(* IEC 61131-3 sources: ml2plc/examples/models/structured_text (part 10) *)

    weights_2 : ARRAY[0..587] OF REAL := [0.015340, -0.219861, -0.051065, 0.087872, 0.001123, -0.000694, -0.000503, -0.080889, -0.021135, -0.014471, -0.082583, -0.025172, 0.069586, 0.000587, -0.088471, 0.003759, -0.014212, -0.039110, -0.007912, -0.105317, -0.021763, 0.126463, -0.041350, 0.108134, -0.142301, -0.053275, 0.007500, 0.120579, 0.091133, 0.103068, -0.006133, -0.082495, 0.034790, 0.002800, 0.014254, 0.050135, 0.050392, -0.065882, 0.073643, 0.079869, -0.165370, -0.153988, 0.109092, 0.031460, 0.038941, -0.087463, -0.087233, -0.123573, -0.001647, 0.004770, 0.048463, -0.043877, -0.184602, -0.074370, 0.166586, 0.231821, -0.353194, 0.011201, 0.023368, 0.060943, 0.075272, -0.042498, 0.053250, -0.100004, -0.036177, 0.065228, -0.023655, -0.016418, -0.006418, -0.172362, -0.131650, 0.045625, 0.096511, 0.126555, 0.121202, -0.064907, -0.098812, -0.091086, 0.010892, 0.012223, -0.059166, 0.035979, -0.151760, 0.028790, 0.081683, 0.051266, -0.099853, -0.051092, 0.055367, 0.050935, -0.059011, -0.033349, -0.019745, -0.141106, -0.147728, -0.164434, -0.113353, -0.053255, 0.023697, 0.071369, 0.115603, -0.270532, -0.017005, 0.015443, 0.033358, -0.027488, -0.120684, 0.053873, 0.046257, -0.048391, -0.013597, -0.155116, -0.101134, -0.222254, 0.105084, 0.104957, -0.208010, -0.081657, -0.136778, -0.070762, 0.148919, 0.151061, 0.138501, 0.115350, 0.039400, 0.091898, -0.109483, -0.207599, -0.054447, 0.127668, 0.008047, 0.087241, -0.038910, 0.138434, -0.038079, 0.070282, 0.095658, 0.048807, -0.081151, -0.133361, 0.009412, -0.027122, -0.098228, 0.001431, 0.004148, -0.083694, -0.036905, -0.212899, -0.099266, -0.054151, 0.010881, -0.082305, -0.021167, -0.016677, -0.138309, -0.079492, -0.045268, -0.012169, -0.016324, -0.059901, 0.029291, 0.037319, -0.106169, 0.072890, 0.053698, 0.036590, 0.031903, 0.081211, 0.046060, 0.124919, 0.117014, -0.103158, -0.081969, 0.141857, 0.110490, 0.008438, 0.045665, -0.042151, -0.082792, -0.089687, 0.003011, -0.079598, -0.013750, 0.011140, -0.033389, 0.000607, 0.054720, 0.044793, 0.059433, -0.049758, 0.003480, 0.032585, 0.099914, 0.124206, -0.103656, -0.036959, 0.191891, -0.166580, 0.032615, 0.068289, -0.002894, 0.153752, 0.186112, -0.195345, -0.026172, -0.075779, -0.150166, 0.066905, 0.193295, -0.375487, -0.153804, -0.064015, 0.001013, 0.051095, -0.055609, -0.045019, -0.076890, -0.054708, -0.006689, -0.066367, 0.086120, 0.139797, -0.050011, -0.067812, -0.047263, -0.073355, -0.003271, 0.015706, 0.020044, -0.025812, 0.092713, 0.059356, 0.027340, 0.108126, 0.188838, -0.104976, -0.027165, 0.083738, 0.040041, 0.159310, 0.142973, 0.100962, -0.057635, 0.104709, -0.046478, 0.050873, 0.025351, -0.109376, 0.011739, -0.063282, -0.068576, -0.007735, -0.119382, 0.145221, -0.087949, -0.001548, 0.079334, 0.050926, -0.020037, -0.015313, 0.046571, 0.032091, 0.023714, 0.049098, 0.043621, 0.065767, -0.121593, -0.144732, 0.087293, -0.020124, 0.165755, -0.049488, -0.192976, -0.057565, -0.115345, -0.055495, -0.078657, 0.070386, 0.053267, -0.047640, 0.089666, 0.074974, 0.047833, 0.104152, -0.039127, 0.127704, -0.117635, 0.009256, 0.057764, -0.018319, 0.044890, -0.124445, -0.081869, -0.128226, 0.073160, -0.069937, 0.090754, 0.040999, -0.061193, 0.026409, 0.119392, -0.038913, -0.081897, 0.050141, -0.041159, 0.018876, -0.029160, 0.061441, 0.084635, -0.047072, 0.062523, 0.081736, 0.012864, -0.124673, -0.040521, -0.031922, 0.010283, 0.007151, -0.035083, 0.061101, 0.118654, -0.023953, -0.013829, 0.030714, -0.167063, -0.041738, -0.014768, -0.060637, 0.029150, 0.043681, 0.069267, -0.066030, 0.016060, 0.030191, 0.072170, 0.120849, -0.083327, -0.090694, -0.027987, 0.023541, 0.067148, 0.139641, 0.111992, 0.115982, -0.002341, 0.013067, -0.113392, -0.151181, 0.086295, 0.008997, 0.108310, 0.012295, 0.020733, 0.024920, -0.047194, -0.007393, -0.027599, 0.150969, 0.041255, -0.072869, -0.231603, -0.078684, -0.006606, -0.022358, -0.011507, -0.054861, 0.048565, -0.117770, 0.037562, -0.101887, -0.217231, -0.177524, -0.162331, -0.325387, 0.103984, 0.039200, -0.041771, 0.006172, 0.062825, -0.139174, -0.098610, -0.065995, -0.047678, -0.009318, 0.107075, -0.006649, 0.059119, 0.087902, 0.003926, 0.023742, -0.024262, -0.018050, 0.007341, 0.009480, -0.122970, -0.021484, 0.124687, 0.030027, 0.096136, 0.053442, 0.014279, 0.038727, 0.068228, -0.029878, 0.026607, 0.088246, 0.138748, -0.166321, -0.035119, 0.030434, -0.057495, 0.037143, -0.085420, 0.031156, 0.004837, -0.115455, -0.013989, 0.165773, 0.007360, 0.120774, -0.095685, -0.203753, -0.112300, -0.139024, 0.004306, -0.041803, -0.030506, -0.033363, -0.031449, 0.092906, 0.227986, -0.103965, 0.010845, -0.128290, 0.097496, -0.021628, 0.017594, 0.054620, 0.088933, 0.056891, -0.002936, -0.038590, -0.048186, -0.021997, 0.106340, 0.017138, 0.079845, 0.036567, -0.064192, 0.034146, 0.052743, -0.004024, 0.135401, -0.092349, -0.039482, 0.036607, -0.113198, 0.036544, 0.077170, 0.046460, 0.094072, 0.058304, 0.084231, -0.093658, 0.080444, -0.094438, 0.026712, 0.042926, -0.037896, 0.031974, 0.018030, -0.045118, 0.039413, -0.087483, 0.054411, -0.109296, -0.120550, 0.081438, 0.039630, 0.131441, 0.016337, 0.018872, 0.038904, 0.024723, -0.125727, -0.003417, 0.113643, 0.012522, 0.023285, -0.022591, -0.082088, -0.102981, -0.128956, 0.016828, 0.053169, -0.013050, 0.047433, 0.119200, -0.020646, 0.082886, 0.121989, -0.094658, -0.060755, 0.019658, -0.020039, 0.056247, 0.054539, 0.134044, 0.104659, 0.135269, -0.109605, -0.042843, 0.008803, 0.033988, -0.264132, -0.142610, -0.095774, -0.150958, 0.018190, 0.003449, -0.089845, -0.132400, 0.022324, 0.100510, -0.288181, -0.014459, 0.059133, 0.074987, -0.005254, -0.103758, -0.007229, -0.006405, 0.006130, 0.046741, 0.116869, -0.032138, 0.051615, -0.051291, -0.050372, -0.068670, 0.011227, 0.032439, 0.064744, 0.039815, -0.046261, 0.007456, 0.054653, -0.076340, 0.076204, -0.009191, 0.110411, 0.126815, 0.058138, -0.038349, 0.037423, 0.073164, 0.105311, 0.107432, -0.038734, -0.004818, 0.013107, 0.024137, -0.005680, 0.019150, 0.033298, 0.097045, 0.108157, 0.044789, -0.004634, 0.055465, 0.016219, 0.151309, 0.033116, 0.036895, 0.003101, 0.089325, 0.030543, 0.060574, -0.338772, 0.009696, -0.068708, -0.048821, 0.097889, 0.163710, 0.087727, 0.021977, -0.192762, -0.018846];
    bias_2 : ARRAY[0..2] OF REAL := [-0.598696, 0.937560, -0.406395];

END_VAR

VAR
    (* Buffer allocation variables *)
    buffer_0 : ARRAY[0..195] OF REAL;
    buffer_1 : ARRAY[0..255] OF REAL;

    (* Temporary computation variables *)
    i : DINT;
    j : DINT;
    sum : REAL;
    max_val : REAL;
    exp_sum : REAL;

END_VAR

(* Layer 0: Fused Linear + RELU *)
FOR j := 0 TO 255 DO
    sum := 0.0;
    FOR i := 0 TO 4 DO
        sum := sum + input_data[i] * weights_0[i * 256 + j];
    END_FOR;
    buffer_1[j] := MAX(sum + bias_0[j], 0.0);
END_FOR;

(* Layer 1: Fused Linear + RELU *)
FOR j := 0 TO 195 DO
    sum := 0.0;
    FOR i := 0 TO 255 DO
        sum := sum + buffer_1[i] * weights_1[i * 196 + j];
    END_FOR;
    buffer_0[j] := MAX(sum + bias_1[j], 0.0);
END_FOR;

(* Layer 2: Fused Linear + SOFTMAX *)
FOR j := 0 TO 2 DO
    sum := 0.0;
    FOR i := 0 TO 195 DO
        sum := sum + buffer_0[i] * weights_2[i * 3 + j];
    END_FOR;
    output_data[j] := sum + bias_2[j];
END_FOR;

max_val := output_data[0];
FOR i := 1 TO 2 DO
    IF output_data[i] > max_val THEN
        max_val := output_data[i];
    END_IF;
END_FOR;

exp_sum := 0.0;
FOR i := 0 TO 2 DO
    output_data[i] := EXP(output_data[i] - max_val);
    exp_sum := exp_sum + output_data[i];
END_FOR;

FOR i := 0 TO 2 DO
    output_data[i] := output_data[i] / exp_sum;
END_FOR;

END_FUNCTION_BLOCK

(* ---- test7_6k.st ---- *)
FUNCTION_BLOCK NeuralNetworkFB

VAR_INPUT
    input_data : ARRAY[0..4] OF REAL;
END_VAR

VAR_OUTPUT
    output_data : ARRAY[0..2] OF REAL;
END_VAR

VAR CONSTANT
    weights_0 : ARRAY[0..399] OF REAL := [-0.204252, 0.095494, -0.178736, -0.051593, -0.154857, -0.111379, -0.197264, -0.143097, 0.109827, -0.097160, 0.012020, -0.049268, -0.066065, 0.005468, -0.112784, -0.022716, -0.225224, -0.191850, -0.006850, 0.088268, 0.127013, -0.051319, -0.177738, -0.065624, 0.153682, 0.155821, 0.040109, -0.174692, -0.286252, 0.062215, -0.175209, -0.111276, -0.147501, -0.127080, 0.122492, 0.111213, 0.028250, -0.187593, 0.149308, 0.140091, 0.112817, -0.082366, -0.154004, 0.019695, -0.076321, 0.047790, -0.005837, 0.106352, -0.126226, -0.091414, -0.224965, -0.021193, 0.065960, 0.078478, -0.162489, -0.177320, 0.118103, -0.118781, -0.258763, -0.167764, -0.097012, -0.191475, -0.225075, -0.097829, -0.133086, -0.161308, 0.068450, -0.142950, -0.218535, 0.051961, 0.024169, -0.169507, -0.262286, 0.029901, 0.048540, 0.027806, -0.189779, 0.069045, 0.117139, -0.010558, -0.032235, -0.086801, 0.151290, 0.170069, 0.043408, -0.094498, -0.177663, 0.095259, -0.083921, 0.266576, -0.232399, 0.088012, -0.144461, 0.013028, 0.218332, 0.118870, 0.049978, -0.108692, -0.017786, -0.028464, 0.071001, -0.202678, -0.007252, 0.046975, -0.022387, -0.176915, 0.184037, 0.138823, 0.117583, 0.033052, 0.015849, 0.231544, 0.199028, -0.026578, -0.236188, 0.131210, -0.105877, -0.087975, -0.089525, -0.271682, -0.310378, -0.190208, -0.103984, 0.021078, -0.061623, -0.223657, 0.115391, -0.052116, -0.091774, 0.111931, -0.085383, -0.115295, -0.241702, -0.144102, -0.001192, -0.097169, -0.177709, -0.113947, -0.007674, -0.135584, 0.123896, 0.092379, 0.005358, -0.157152, -0.059988, -0.012534, 0.034736, -0.043048, 0.057696, -0.238518, 0.035371, -0.093588, 0.167829, -0.046709, 0.036370, -0.003444, -0.106658, 0.028076, 0.151991, 0.154167, -0.017135, -0.263429, 0.026569, -0.116189, -0.091898, 0.047045, 0.267170, 0.114090, 0.116855, 0.032118, 0.099443, 0.013459, 0.247495, -0.047596, -0.170523, -0.138334, -0.014806, 0.093128, -0.113583, -0.042853, -0.078199, 0.216203, 0.089752, -0.194084, -0.181997, 0.131227, -0.069781, 0.133463, -0.154973, 0.009000, -0.012056, -0.165474, 0.081740, 0.099855, -0.149436, -0.029881, -0.055397, 0.210030, -0.245871, 0.129955, 0.110984, 0.270213, 0.000066, -0.234064, -0.167355, -0.006196, -0.161614, -0.083333, -0.230470, -0.085398, -0.155489, 0.196806, 0.059367, 0.177773, -0.031812, -0.105303, 0.169684, 0.096922, -0.081472, 0.044204, -0.176394, -0.252753, -0.084089, 0.174208, 0.011128, 0.036618, 0.039985, 0.063442, 0.014899, 0.025740, -0.126109, 0.051767, 0.112909, 0.030818, 0.068933, 0.024684, -0.106318, -0.005054, -0.144284, -0.256852, -0.164291, -0.133206, -0.210012, -0.101632, 0.222082, 0.153257, -0.192512, 0.005971, -0.123604, -0.264094, -0.027056, -0.013892, -0.236922, 0.115783, 0.095674, 0.181820, 0.094948, 0.002586, -0.087751, -0.234015, -0.217941, -0.202149, -0.182678, -0.162661, -0.103708, -0.300429, -0.038539, -0.114616, -0.039287, -0.323055, -0.037187, 0.185280, -0.134350, -0.202214, -0.095785, -0.238161, 0.248820, -0.025541, 0.153553, -0.146549, 0.025226, -0.124733, -0.153933, -0.057788, 0.112253, 0.171774, -0.055901, 0.100347, -0.016596, 0.038081, 0.060529, -0.211000, 0.010525, -0.175179, -0.266535, 0.149374, -0.227717, 0.025317, 0.156851, 0.099082, 0.142311, -0.009360, 0.116468, 0.063573, 0.171788, 0.104363, -0.112531, 0.109297, 0.087755, -0.007313, 0.042170, 0.011677, -0.244264, -0.025654, -0.082018, -0.040680, -0.066031, 0.099246, -0.016522, -0.033168, -0.102887, -0.139828, -0.135602, -0.001694, -0.159093, -0.118193, 0.253445, -0.227600, 0.115132, -0.149348, -0.024129, -0.094190, -0.174122, 0.091905, 0.084444, -0.253624, 0.046840, 0.005839, 0.162217, -0.263061, 0.010626, 0.172488, 0.044317, 0.030137, 0.082965, -0.289103, -0.425034, 0.089364, 0.139634, -0.374789, 0.002438, -0.053035, -0.205200, 0.042774, 0.083738, 0.165071, -0.181691, -0.060783, -0.208866, -0.016353, -0.150721, 0.082961, -0.194339, -0.103480, -0.062981, 0.183148, -0.146493, -0.192516, 0.006207, 0.166178, 0.119890, -0.161796, -0.046662, -0.139639, 0.107740, 0.150401, -0.042296, 0.020544, -0.142547, 0.079611, 0.168141, 0.162479, -0.125809, -0.131995, 0.147326, 0.206230, 0.039064, -0.003743, -0.201281, 0.075811, 0.106736, -0.157088, 0.096469, 0.149164, -0.048443, -0.147991, 0.003754, -0.211540, -0.015394, -0.123360];
    bias_0 : ARRAY[0..79] OF REAL := [0.085009, 0.139520, 0.248067, 1.399861, 0.583598, 0.015434, -0.202390, 0.740568, -0.902567, 0.016522, -0.292847, 1.752811, -0.063338, -0.564435, -1.102493, -0.004024, -0.597225, 0.046091, 0.423281, 0.308277, -0.198749, 0.191307, -0.275388, -0.046908, -0.389957, 0.456703, 0.444849, -0.885773, 0.015246, 0.438173, 0.310576, -1.156887, 0.283457, -0.324643, -0.165189, -0.746600, 0.758963, -0.005614, -0.150126, 0.284105, -0.379746, 0.854058, -0.107690, 0.052858, -0.034767, -0.935268, -0.085336, 1.113907, -0.062266, -0.710800, -0.218181, 0.473975, 0.306379, 0.051084, -0.381713, 0.449957, 0.295188, -0.428395, 0.386686, -0.302978, -0.218029, -0.006667, 0.249048, 0.384831, -1.063448, -0.870574, -0.613569, -0.747093, -0.019498, -0.541172, -1.064162, 0.472992, 0.204574, -0.857920, -0.625336, -0.146532, -0.007889, -0.730171, -0.376830, -0.026634];

    weights_1 : ARRAY[0..4799] OF REAL := [-0.187495, -0.043826, 0.011639, 0.068499, -0.019446, 0.115631, -0.047638, -0.110905, 0.095464, -0.000825, -0.147106, -0.138385, 0.173698, -0.115326, 0.005790, -0.077005, 0.183801, -0.196797, -0.004029, -0.178881, 0.095461, -0.234334, 0.116176, 0.020930, 0.100273, -0.069382, 0.012484, -0.061318, 0.076773, -0.161382, -0.212827, -0.106095, -0.170268, -0.227658, -0.157359, -0.001001, 0.019196, 0.052587, -0.065633, 0.121859, -0.043743, 0.056348, -0.200779, 0.011906, -0.185246, 0.005645, -0.224972, -0.078873, 0.012620, -0.098199, -0.035988, -0.043461, -0.058674, -0.026206, 0.058788, -0.126039, -0.214524, -0.215762, -0.047320, -0.167665, 0.081893, -0.181390, 0.147489, -0.050866, -0.159085, 0.025241, -0.075018, 0.080488, -0.144720, -0.183416, -0.000486, 0.277692, -0.025934, -0.091180, 0.135423, -0.071436, -0.206965, -0.032235, -0.070909, -0.118695, 0.120077, -0.224050, -0.086073, 0.058597, -0.003604, -0.190653, 0.187794, -0.105244, -0.139862, 0.095354, -0.079105, -0.049326, -0.180191, 0.046015, -0.008404, -0.009414, 0.007191, -0.167950, 0.064259, 0.028046, -0.065026, 0.002607, 0.055868, -0.016474, 0.038395, -0.073723, -0.001131, -0.097771, 0.086923, 0.060480, 0.102652, 0.151700, -0.249111, -0.000081, -0.115305, 0.119442, -0.017911, -0.276544, -0.195153, 0.023084, 0.061307, -0.149912, 0.126201, 0.077160, 0.147664, 0.135438, 0.179792, -0.136279, 0.128259, -0.029156, -0.105667, -0.013778, 0.067171, -0.212397, 0.135022, -0.092745, -0.212069, -0.083156, -0.273877, -0.080802, -0.036298, 0.074901, -0.197178, 0.189450, -0.212966, 0.089309, 0.201708, -0.157652, 0.104825, -0.088819, -0.017402, -0.200047, -0.095955, 0.102139, 0.042738, -0.085193, -0.087002, -0.084559, 0.014232, -0.160413, -0.342999, -0.172071, 0.030429, -0.141189, -0.242259, -0.189519, 0.141134, -0.151873, -0.033610, -0.155085, 0.096499, -0.170400, -0.030843, -0.192798, 0.082588, -0.197594, -0.127308, -0.215119, -0.164729, -0.082233, -0.329844, 0.368244, -0.284488, -0.291019, -0.331445, 0.198686, -0.097576, -0.033210, 0.217893, 0.111894, -0.030753, -0.229657, 0.127646, -0.247362, 0.004571, -0.221431, 0.197898, 0.003611, 0.001089, 0.217739, 0.009284, -0.169147, -0.171246, -0.217403, -0.194864, 0.208354, -0.316288, -0.209805, -0.538319, 0.125899, -0.174896, -0.237079, 0.022632, 0.071399, 0.183040, -0.119043, -0.077857, -0.037180, 0.391291, 0.080994, 0.094256, -0.231882, 0.044936, 0.172367, -0.197255, -0.202964, -0.189238, 0.088037, 0.016176, 0.049230, 0.086076, -0.165083, -0.123050, -0.217327, -0.104082, -0.184468, -0.084095, -0.192575, -0.003610, 0.003037, -0.109199, 0.129669, -0.121035, -0.062529, -0.063750, 0.104687, 0.028781, -0.149673, 0.198580, 0.131386, 0.071709, -0.227315, 0.138179, -0.009123, 0.102321, -0.095555, 0.094151, 0.123000, 0.224575, -0.096633, 0.042278, 0.084082, 0.031284, -0.107486, 0.016887, -0.039989, 0.009479, -0.112127, -0.227535, 0.007071, -0.043445, -0.166035, 0.115495, -0.269776, 0.124071, -0.072062, -0.180874, -0.140957, 0.158938, -0.171277, -0.151687, 0.004736, -0.133418, 0.071863, -0.123936, -0.008774, -0.073201, -0.059242, -0.054432, 0.027825, -0.161739, -0.079946, 0.093769, 0.128523, 0.043888, -0.155475, -0.230641, 0.122559, 0.076405, -0.181072, -0.127761, 0.012384, 0.021831, -0.244387, 0.085400, -0.134273, -0.205303, -0.012499, 0.001737, 0.098550, -0.193665, 0.050139, 0.092846, -0.051853, 0.048240, 0.039286, 0.149299, -0.087487, 0.155728, 0.110941, 0.075036, -0.149393, 0.069146, 0.188267, -0.152000, -0.172031, 0.024997, -0.087718, 0.050184, -0.153210, 0.046277, -0.180275, -0.025535, -0.116391, 0.104334, 0.018564, -0.028917, -0.084740, -0.136146, -0.100181, 0.038304, 0.091499, -0.064747, 0.160913, -0.017199, -0.147531, -0.109603, -0.032457, 0.097940, -0.100716, -0.059666, -0.061391, 0.088145, -0.192598, -0.125311, -0.157310, 0.002378, 0.121867, 0.102271, 0.080352, -0.057906, 0.063848, 0.019965, -0.227923, 0.051208, 0.088724, 0.149698, 0.064482, -0.033688, -0.202038, 0.055623, -0.142244, 0.118062, 0.013894, -0.217208, 0.125276, -0.085431, -0.050093, -0.078770, -0.127041, -0.181141, 0.038965, -0.253101, -0.069012, -0.148941, 0.028103, -0.097699, -0.128741, -0.147791, 0.149346, 0.024986, 0.058569, 0.143465, 0.145976, -0.067909, -0.015331, -0.043340, -0.096023, 0.123826, 0.016238, -0.173743, -0.066383, 0.091369, -0.029829, 0.159701, -0.052570, -0.188634, 0.033418, -0.043469, 0.226051, -0.138364, -0.055090, 0.100096, 0.054385, -0.082675, 0.052667, -0.174938, -0.010745, -0.130078, 0.125440, -0.065375, 0.079887, -0.045133, -0.048312, -0.037418, -0.081846, 0.128402, -0.121171, -0.021942, -0.143802, -0.240385, -0.098094, 0.214161, -0.048066, -0.104972, 0.177667, -0.027555, 0.199294, -0.277881, -0.103592, -0.101064, -0.111686, -0.052772, 0.002445, -0.221140, 0.200714, -0.029648, -0.351862, 0.087262, 0.149245, -0.019061, -0.170681, 0.079724, -0.139517, -0.080832, -0.183112, -0.155987, 0.111392, -0.012468, -0.261954, -0.013893, -0.140637, -0.064067, 0.087971, -0.098510, -0.073594, 0.139888, -0.085039, 0.040758, -0.128766, 0.263592, -0.257286, -0.202891, 0.100467, -0.010248, 0.014490, 0.076027, -0.041766, -0.131794, -0.181699, 0.141993, 0.089453, -0.191971, 0.038637, 0.071693, 0.041796, 0.073103, 0.145141, -0.148769, 0.095703, -0.006099, 0.053828, -0.166412, 0.109511, 0.111218, 0.062706, 0.039294, 0.024273, -0.008815, -0.122314, 0.041015, -0.064941, -0.049589, 0.162990, 0.170278, -0.122815, 0.145788, 0.033580, 0.010933, 0.020278, 0.165807, -0.145881, 0.200069, 0.132890, -0.225906, 0.102775, 0.112111, -0.110968, -0.327020, -0.063996, 0.018829, -0.105115, -0.035790, -0.111621, -0.161010, -0.136633, 0.132319, -0.232511, 0.068281, -0.190410, -0.280823, 0.037700, -0.036999, -0.202194, -0.009511, -0.062345, 0.223302, 0.224884, -0.037151, 0.133080, -0.105688, 0.104093, -0.044832, -0.119623, -0.100510, -0.010594, -0.177663, -0.143772, -0.129429, -0.155730, 0.074013, 0.203130, -0.168618, 0.197457, -0.075762, 0.002407, -0.127743, -0.027171, 0.040017, -0.164665, -0.133451, -0.093815, 0.045166, -0.370300, -0.136726, -0.057434, -0.196779, -0.123197, 0.054104, -0.153149, -0.058581, -0.200545, -0.337820, -0.223224, -0.084699, 0.068145, -0.023780, -0.075253, 0.104862, 0.092775, 0.252090, -0.182647, -0.060455, 0.193314, 0.155096, 0.017778, -0.041913, 0.080495, 0.250374, -0.062116, -0.031334, -0.091330, -0.297533, 0.067413, -0.122810, -0.020310, 0.102734, -0.089518, -0.069400, -0.252473, 0.055755, -0.067582, 0.124237, -0.105892, -0.185992, 0.084798, -0.008859, -0.000417, -0.200312, -0.077944, 0.154457, 0.008785, 0.210066, 0.124764, 0.010203, 0.027909, -0.020809, -0.104830, -0.241088, 0.075725, -0.243988, -0.073502, -0.150011, 0.042442, -0.016308, -0.053375, 0.203016, -0.189589, -0.147536, -0.000456, 0.010458, -0.016922, -0.023293, -0.229019, -0.031755, -0.225682, 0.136042, 0.163329, -0.145518, -0.137362, -0.158810, -0.153608, -0.119005, -0.139013, 0.068120, -0.178356, -0.217439, 0.098411, 0.179662, 0.050977, -0.148974, 0.173078, 0.154025, -0.222811, 0.095003, 0.026945, -0.065555, -0.157365, -0.148347, 0.083820, 0.203749, 0.276060, -0.130301, -0.441604, 0.101892, 0.325627, -0.175195, 0.033774, 0.197460, -0.021086, -0.054220, -0.115699, -0.068489, -0.046554, -0.156783, 0.161611, -0.049137, 0.005860, 0.193781, 0.370352, -0.216234, 0.350976, 0.064933, -0.356365, 0.030951, 0.310719, -0.269228, 0.000328, -0.685306, 0.092410, -0.057984, -0.234432, -0.157181, -0.054908, 0.119585, 0.055568, 0.033589, 0.070298, 0.151600, 0.000321, 0.203942, -0.184519, -0.196852, 0.020012, -0.127641, -0.136458, 0.095097, -0.156321, -0.046661, -0.126675, 0.034023, -0.435073, -0.248280, 0.038863, 0.051302, -0.121698, -0.248643, -0.253840, -0.235557, -0.057713, -0.165379, -0.072123, 0.012063, 0.179261, -0.079980, -0.109507, 0.061432, 0.149497, -0.070263, 0.063627, -0.203408, -0.054263, 0.041969, 0.093557, 0.035906, -0.075950, -0.132530, 0.160581, -0.093528, -0.193797, -0.149616, 0.081809, 0.132168, -0.055765, -0.226921, 0.052611, -0.019008, -0.206362, 0.196463, 0.058143, 0.139270, -0.182240, -0.077353, 0.126875, 0.019908, -0.178625, 0.207289, 0.023789, -0.110765, -0.042038, 0.090671, -0.010270, 0.088242, -0.078280, 0.027414, 0.024751, -0.053083, -0.111664, 0.145266, 0.045896, -0.106047, 0.028589, 0.126394, -0.073975, 0.016951, -0.114771, 0.058699, 0.138664, -0.111792, 0.102104, -0.085657, 0.025535, -0.077525, 0.176288, 0.007275, 0.013041, -0.182064, -0.008665, 0.010742, -0.063345, -0.170987, 0.118484, 0.086599, -0.138879, 0.062084, 0.093707, -0.211441, -0.210389, 0.109447, 0.009178, 0.111142, 0.057708, -0.107554, -0.097098, -0.050753, -0.119869, 0.065488, -0.195523, 0.125473, -0.162880, 0.067520, -0.057914, 0.067633, -0.128362, -0.041456, -0.151078, -0.239852, -0.046787, -0.046040, -0.085033, -0.027876, -0.050788, -0.175431, 0.021347, 0.129480, -0.202736, -0.211963, -0.121893, -0.053449, 0.174972, -0.090305, -0.027340, 0.184640, 0.018241, -0.146348, -0.088299, -0.200020, 0.179131, -0.156040, 0.247591, -0.018738, -0.167393, -0.018119, 0.166582, 0.036737, -0.323502, -0.125462, -0.074257, -0.227693, -0.127879, 0.074497, 0.171681, -0.178597, -0.016256, 0.165335, 0.142548, -0.065136, -0.057195, 0.137034, -0.103093, -0.057882, -0.106992, -0.082292, 0.014769, -0.131339, -0.122740, 0.221346, 0.050323, -0.115536, -0.161429, -0.121929, -0.141410, -0.200174, -0.131279, -0.070172, -0.001654, -0.054385, -0.203309, -0.174031, -0.044717, -0.023823, -0.195514, 0.097579, -0.299280, 0.071825, -0.120568, 0.121904, 0.022071, 0.004942, -0.093524, -0.047500, 0.108046, 0.027347, 0.109685, -0.057970, 0.069021, -0.106463, 0.151177, -0.178336, -0.105863, 0.119959, -0.270658, 0.072922, -0.081703, -0.126428, -0.064988, 0.119859, -0.148058, -0.121758, -0.124044, -0.181647, 0.103696, -0.059793, 0.009263, -0.067097, -0.157507, -0.210798, -0.108414, 0.015803, 0.100605, 0.001284, 0.092993, -0.114392, -0.198128, -0.107984, -0.135560, -0.212594, -0.122395, 0.051632, 0.120981, 0.036958, -0.088017, 0.048821, 0.105228, 0.039687, -0.000940, 0.117730, 0.094232, 0.097422, -0.162968, -0.207689, -0.235039, -0.020052, 0.003264, 0.066222, -0.007693, 0.112790, 0.004400, -0.170587, -0.007529, -0.092564, -0.071948, 0.098179, -0.173899, -0.189986, 0.082992, 0.049693, -0.084597, -0.022957, -0.112488, -0.177351, -0.074619, 0.043721, 0.081083, 0.056966, -0.054530, 0.167706, 0.092779, 0.038886, 0.052530, 0.175779, 0.062225, 0.067869, -0.150979, -0.026430, 0.041959, 0.159334, 0.014994, -0.132202, -0.203469, -0.166479, -0.001058, 0.032094, 0.102088, -0.026257, 0.108982, -0.197880, -0.186123, -0.210913, -0.013239, 0.133741, 0.024038, 0.035955, 0.009580, -0.220388, -0.093084, -0.115529, 0.113373, -0.179200, 0.023569, 0.092303, -0.057884, -0.182442, -0.125423, 0.135616, 0.148641, 0.001794, 0.053828, -0.009687, -0.061003, -0.109162, -0.094053, 0.085367, -0.054325, 0.003022, 0.109594, 0.150069, -0.100455, -0.027854, -0.045738, 0.104897, -0.098767, -0.052057, -0.014638, -0.046503, -0.088066, -0.196605, -0.111631, 0.106046, 0.108629, -0.197552, -0.149193, 0.109600, -0.177730, 0.155000, 0.139756, 0.156765, 0.093107, -0.180579, -0.112168, 0.171606, -0.097841, 0.105849, 0.202372, -0.155509, 0.025837, -0.097935, -0.208450, 0.082403, -0.195167, -0.064462, -0.168772, 0.181297, 0.110526, -0.082017, 0.062444, -0.085259, 0.031226, 0.195569, 0.136555, -0.089863, 0.044305, -0.224308, 0.062433, -0.141740, -0.045204, 0.123520, 0.036962, -0.120294, -0.095129, -0.174097, 0.052688, 0.011449, -0.176074, -0.065089, -0.038276, 0.090562, 0.076366, -0.075167, 0.061729, 0.038455, 0.053242, -0.193444, 0.101651, 0.087634, 0.092511, -0.064193, -0.245658, 0.044015, 0.012871, -0.013168, -0.006454, 0.071112, 0.025509, 0.054529, 0.065311, 0.056310, -0.180449, -0.039958, 0.048537, -0.051643, -0.102219, 0.113807, -0.057327, 0.046546, -0.151255, -0.077736, -0.020588, -0.113985, 0.169675, 0.052531, 0.048476, 0.012000, -0.042925, 0.130053, -0.008425, 0.126301, -0.005038, -0.050381, 0.101160, -0.260447, 0.032194, -0.186597, 0.099273, -0.066057, 0.020545, -0.196886, -0.214360, 0.135345, -0.000402, 0.039084, -0.102168, 0.155453, -0.083347, -0.293784, -0.056957, -0.158940, -0.024392, 0.012893, 0.016886, 0.001811, 0.142059, -0.177070, 0.081076, -0.177536, -0.008914, 0.128194, 0.078825, -0.001006, -0.140982, 0.025296, 0.312801, -0.009939, -0.234129, 0.156600, 0.074625, 0.204806, 0.080406, -0.245319, -0.007829, -0.125331, -0.077263, -0.269901, 0.007388, 0.072491, 0.187339, -0.021148, -0.141481, -0.151382, -0.091537, -0.024638, -0.063637, -0.002112, -0.242162, 0.068506, -0.194093, 0.147597, -0.224350, -0.109162, -0.248442, -0.281311, 0.099040, -0.114785, -0.153094, -0.143746, 0.119874, 0.245667, -0.073279, -0.106678, 0.070350, -0.065192, 0.189557, -0.053012, 0.006938, -0.168214, -0.159039, 0.099331, 0.042333, -0.011618, 0.036502, -0.046085, 0.022646, -0.169739, -0.134299, -0.147109, -0.055030, -0.207480, 0.034523, -0.053364, -0.170573, 0.062128, -0.108211, -0.087569, 0.096130, 0.105775, -0.076363, -0.149795, 0.111862, 0.064433, 0.100011, 0.005322, 0.012295, 0.044367, 0.038804, 0.036462, -0.009752, 0.027189, -0.112119, -0.197054, -0.207718, 0.029751, -0.157544, 0.098411, -0.107287, -0.004124, 0.110229, 0.022413, 0.077564, 0.045048, 0.160432, 0.136350, -0.067685, 0.121371, -0.045504, 0.001140, 0.092194, 0.093704, -0.197313, -0.053982, 0.058188, 0.107029, -0.190503, 0.017645, 0.056198, -0.165373, -0.188030, 0.177592, 0.143248, 0.150138, 0.040068, 0.016359, -0.087664, 0.029084, 0.063598, 0.117892, -0.012894, -0.281147, 0.019644, 0.077236, -0.102193, 0.001728, -0.201237, -0.046811, 0.187137, -0.088159, 0.098611, -0.190801, 0.099519, 0.009386, -0.009936, -0.095895, 0.043072, 0.069656, -0.116856, -0.044185, 0.024672, 0.066147, 0.123219, 0.026984, 0.061291, -0.161035, -0.117871, -0.023781, 0.020670, -0.044119, -0.150813, 0.119473, 0.264945, -0.078791, -0.174729, -0.082116, 0.065382, -0.160124, 0.058964, -0.173368, -0.063958, 0.150073, 0.137277, 0.040349, -0.121023, 0.102109, 0.155909, 0.029025, 0.055306, -0.196372, 0.094951, 0.105758, -0.108173, -0.029256, -0.069724, -0.036958, 0.102471, 0.089850, 0.085119, -0.179385, 0.077873, -0.058101, -0.064385, 0.122941, -0.197724, 0.096621, 0.136942, -0.086460, 0.097450, -0.194683, 0.020468, -0.091201, -0.163263, -0.060383, -0.122360, 0.063817, -0.261001, -0.151872, -0.203316, -0.127345, -0.096171, -0.023894, 0.197431, -0.225454, -0.240749, -0.317417, -0.079323, 0.065090, 0.019849, -0.136263, -0.136703, 0.062078, 0.071355, -0.182125, 0.067118, -0.270489, 0.055133, -0.003778, 0.114173, 0.067716, -0.277999, -0.202380, 0.065272, 0.003847, -0.084694, -0.207460, 0.017935, -0.121946, 0.137768, 0.094442, -0.092968, -0.075586, 0.096753, -0.023769, 0.014763, 0.174060, -0.227682, 0.084332, -0.081958, -0.134817, -0.000166, 0.192078, 0.040887, -0.001630, 0.113297, -0.197617, 0.027211, 0.052274, -0.180139, 0.149111, 0.130356, -0.226361, 0.016953, -0.122692, -0.156576, -0.054064, -0.193463, -0.185229, -0.221918, 0.140038, -0.054511, 0.108777, -0.208394, 0.041422, -0.250061, -0.144061, 0.000987, -0.121394, 0.086455, 0.068661, 0.077966, 0.138036, -0.093587, -0.191712, 0.118125, -0.019484, -0.014273, -0.059302, -0.104286, -0.116784, 0.075291, 0.169043, 0.001548, -0.184765, -0.006782, 0.022824, -0.003976, -0.051564, 0.067487, -0.070492, -0.094790, 0.153426, 0.145733, -0.204557, 0.058039, 0.108285, -0.170155, 0.095073, -0.146102, 0.164169, -0.186476, 0.024414, -0.196119, 0.110557, -0.013596, 0.146735, 0.045880, -0.001961, -0.210447, -0.078950, -0.105805, 0.176049, -0.057586, -0.258445, 0.050336, -0.084662, -0.126641, 0.047383, -0.157251, -0.181100, -0.077797, -0.014061, -0.025577, 0.010956, -0.064073, 0.071510, -0.145995, -0.134231, 0.040794, -0.079272, -0.038888, -0.016440, 0.173860, 0.125972, 0.171500, -0.254024, -0.140350, 0.117999, -0.067682, -0.000752, 0.107778, 0.023448, -0.180043, 0.120349, 0.025010, 0.013541, -0.106484, 0.171297, 0.058092, -0.126303, 0.146605, -0.118698, -0.101074, -0.209394, -0.081997, -0.097325, -0.073534, 0.041903, -0.160915, -0.086830, -0.246047, 0.146267, -0.093346, 0.022996, 0.114033, -0.071188, 0.262760, 0.121509, -0.149237, -0.213894, -0.046132, 0.196951, -0.148721, -0.043823, 0.021680, -0.187718, -0.106041, 0.122252, -0.202239, -0.211710, 0.107129, -0.178040, -0.001868, -0.028487, 0.104841, -0.194258, 0.066877, -0.068969, 0.029807, 0.080136, -0.202076, -0.035068, 0.045806, 0.055710, -0.255747, -0.077842, -0.121811, 0.164499, 0.018934, -0.073491, 0.005038, 0.249075, 0.018043, 0.064148, -0.181961, 0.010560, -0.117548, -0.058183, -0.035022, -0.194345, 0.039141, -0.096355, 0.004603, 0.022892, -0.181091, -0.052832, -0.084987, -0.114381, -0.116218, -0.225355, 0.091435, -0.083195, -0.018672, -0.082354, -0.062302, -0.058156, 0.044570, 0.188819, -0.030222, 0.004905, -0.158938, 0.195750, 0.071720, -0.031885, -0.001187, -0.228501, 0.050306, -0.205469, -0.032645, 0.106419, 0.074064, -0.026300, -0.186675, -0.264539, 0.215900, -0.332340, -0.043278, -0.206134, 0.044834, 0.109163, -0.102909, -0.072938, -0.364193, -0.196215, -0.007963, 0.026792, -0.134129, -0.057963, 0.072873, 0.065697, -0.271673, 0.064010, -0.008266, 0.074413, -0.266393, -0.036302, 0.079263, -0.060772, -0.018792, 0.137687, -0.104393, -0.152897, -0.242089, 0.106164, 0.018856, 0.092918, -0.275230, -0.063488, 0.090247, -0.059361, -0.266099, -0.046778, -0.055142, -0.022777, 0.084627, -0.170351, -0.013962, -0.222389, -0.151188, 0.148962, -0.087542, 0.185998, -0.177688, -0.097772, -0.079313, -0.150211, -0.164873, -0.158232, 0.217011, -0.160489, -0.116968, -0.091767, 0.116603, 0.011526, -0.153908, -0.067538, 0.168542, -0.178588, 0.082390, 0.018650, 0.039973, -0.025669, 0.168206, -0.248549, 0.149303, -0.160598, 0.069041, -0.183907, -0.049261, 0.160879, -0.095732, -0.165781, -0.080461, 0.055374, 0.016760, -0.174546, 0.081962, -0.036502, 0.158612, 0.032619, 0.049739, 0.027940, 0.224843, 0.073671, -0.041689, 0.230666, 0.145157, -0.234841, -0.176481, -0.095837, 0.125010, 0.063278, -0.230302, 0.063268, -0.027022, 0.111030, 0.053486, 0.027500, 0.140594, -0.134408, 0.103652, -0.051922, 0.012637, -0.181476, -0.019460, -0.029901, -0.032062, 0.172354, 0.148283, 0.215879, -0.142901, -0.119957, -0.053013, 0.112965, -0.258184, -0.051066, -0.264954, 0.190482, -0.189949, 0.010940, -0.095231, 0.008937, -0.040283, -0.059043, -0.015149, -0.015143, 0.141878, 0.109967, -0.042080, -0.157305, 0.097915, -0.108920, 0.104729, 0.194386, 0.011276, -0.019095, -0.084019, 0.146113, -0.152649, 0.198303, -0.201287, -0.137585, 0.035677, -0.061117, 0.176087, 0.160562, -0.230831, -0.028126, -0.215707, -0.040773, -0.019594, 0.077786, -0.099227, -0.115451, -0.063161, -0.084506, 0.285519, -0.030241, 0.168914, 0.020630, 0.029172, -0.202726, 0.104421, -0.053312, -0.039889, 0.052079, -0.062510, -0.130882, -0.040990, -0.278632, -0.058964, 0.217417, -0.121801, -0.096731, 0.087152, -0.022312, -0.172589, -0.263482, -0.193324, 0.004411, 0.121928, 0.159931, -0.192278, 0.132315, -0.214687, -0.049484, -0.008205, 0.018524, 0.133953, -0.040444, 0.056558, 0.015706, 0.325216, 0.000640, 0.075307, 0.035595, 0.113399, -0.202202, -0.025153, 0.167535, -0.239881, -0.219585, -0.111719, -0.107923, -0.149904, -0.252613, -0.034304, -0.084333, -0.187109, 0.063899, 0.143530, -0.070666, 0.132294, 0.051739, 0.147802, -0.104738, 0.129664, 0.014652, 0.044681, -0.125330, -0.207789, -0.042319, -0.165956, -0.203115, -0.044789, -0.205011, 0.000517, 0.021081, -0.119809, -0.210937, -0.231928, 0.087419, 0.205960, -0.027473, -0.228470, -0.094027, -0.064081, 0.147182, -0.185475, 0.131948, 0.100349, 0.009282, 0.114615, 0.140396, -0.116940, 0.072523, -0.241860, -0.108013, -0.142000, -0.072000, 0.089677, 0.137196, 0.062616, 0.121207, -0.232016, 0.090843, 0.070410, 0.139417, -0.026856, 0.146321, -0.294664, -0.032348, 0.319110, -0.002944, -0.067224, -0.092913, -0.150887, -0.212212, 0.031102, -0.085811, 0.014206, -0.144119, -0.058346, 0.019250, 0.018418, -0.186849, -0.072161, 0.001996, 0.103666, -0.258730, -0.081637, 0.055279, 0.061815, -0.044559, -0.113122, -0.044066, -0.162221, -0.141151, 0.096907, -0.115250, 0.062262, 0.005065, 0.015412, 0.081220, -0.297356, 0.064133, 0.044118, 0.015685, -0.144599, -0.076847, -0.087228, -0.168556, -0.226387, -0.249636, -0.024162, -0.182325, 0.016776, -0.238902, -0.135556, -0.086752, -0.115952, 0.040745, -0.122256, -0.102772, -0.191892, -0.274205, 0.066162, 0.048205, -0.064058, -0.192005, 0.120239, 0.191195, 0.196010, -0.017396, -0.049525, 0.061457, -0.080446, -0.015556, -0.170852, -0.127559, 0.258399, -0.089019, 0.126596, -0.235834, -0.115058, -0.102991, 0.116196, 0.150089, -0.147114, -0.097072, -0.167377, -0.093958, -0.187377, -0.132066, -0.089605, -0.180094, -0.014606, -0.072250, -0.202879, -0.002921, 0.046777, 0.096036, -0.160877, -0.198220, 0.046167, 0.014711, -0.258481, -0.002196, 0.044809, 0.085482, -0.024420, 0.037063, -0.018678, -0.067966, -0.085948, 0.078864, -0.201114, 0.128085, -0.145813, 0.007271, 0.039512, -0.028435, -0.018339, 0.139499, -0.003059, -0.099800, -0.061026, -0.084604, -0.164472, -0.100570, -0.169849, -0.037404, -0.194296, 0.068681, -0.011228, 0.059797, 0.134118, -0.200450, 0.131266, 0.008578, -0.032415, 0.125618, -0.183185, -0.186559, -0.059436, 0.039473, -0.133920, -0.179227, 0.156785, -0.167550, -0.090492, 0.055735, 0.129721, -0.109047, 0.164852, 0.055422, 0.065316, -0.189822, 0.012060, -0.117954, 0.014381, 0.158313, -0.189159, 0.142768, -0.144892, -0.116591, -0.005984, 0.124853, -0.026583, -0.166240, -0.083795, -0.123045, 0.122757, -0.037477, 0.092098, -0.148620, 0.038476, 0.152449, -0.098045, -0.094949, -0.145768, 0.081120, 0.032547, 0.132474, 0.135196, -0.257294, -0.163471, -0.075842, 0.216315, 0.079247, 0.066841, -0.054610, 0.080234, 0.023575, -0.091794, -0.154834, -0.053194, -0.028051, -0.130317, -0.114688, -0.102097, -0.054053, 0.071980, -0.149434, -0.025769, -0.159231, 0.136723, 0.069798, -0.142915, -0.204482, 0.013283, 0.165752, 0.048956, -0.071522, 0.014189, -0.034166, 0.140926, -0.063779, -0.189843, -0.093377, 0.089115, -0.053616, -0.139420, -0.037278, 0.143302, -0.117698, -0.054848, 0.127853, 0.055342, 0.152365, -0.160254, -0.059313, 0.100204, -0.156020, -0.004533, -0.169456, 0.076558, 0.115337, 0.033748, -0.130311, 0.001136, -0.053222, -0.189011, -0.052963, -0.170158, -0.044768, -0.229454, -0.088228, 0.161163, -0.254016, -0.079255, 0.109965, -0.044888, 0.111780, -0.214687, 0.055047, -0.118845, -0.152920, 0.182037, -0.064142, -0.169884, -0.003040, -0.184904, -0.064518, 0.088405, -0.147685, 0.088867, -0.048795, -0.109284, -0.187385, 0.202099, -0.078681, -0.135884, 0.066514, -0.027167, -0.049248, 0.013263, 0.001392, 0.114698, 0.153221, -0.056513, 0.110682, -0.002497, 0.033449, 0.093565, -0.013117, 0.192191, 0.155546, 0.047371, -0.140575, -0.127799, -0.017932, 0.113502, -0.065293, -0.165022, -0.168184, -0.210941, 0.011351, -0.077979, -0.032503, -0.211552, 0.114545, -0.002053, 0.099328, -0.012842, -0.041377, 0.011279, -0.033605, 0.080875, 0.134533, 0.134824, -0.148507, -0.144622, -0.128805, -0.022675, 0.114730, 0.066712, -0.066104, 0.027683, -0.008968, 0.165856, -0.105824, 0.166434, 0.188111, -0.110221, -0.230624, -0.142589, -0.026202, -0.129956, 0.042155, 0.077495, 0.151450, -0.172573, -0.138375, 0.058228, 0.143052, -0.003161, -0.229277, -0.063510, -0.143647, 0.146517, -0.045903, -0.177465, -0.110375, -0.034529, 0.170249, -0.050045, -0.115385, 0.174185, -0.046401, 0.002193, 0.028995, -0.271681, 0.218660, 0.126515, -0.230110, 0.000361, -0.160436, 0.005971, -0.344556, 0.131244, -0.051877, -0.006286, 0.057548, -0.068816, 0.211492, -0.095057, -0.199010, 0.054005, -0.149013, -0.353793, -0.120430, -0.039355, -0.024089, -0.194303, -0.085727, 0.117557, 0.040830, -0.063834, 0.093352, 0.110169, -0.024051, 0.009023, -0.119322, -0.203330, -0.208702, -0.160522, -0.129267, -0.150143, 0.045876, -0.129271, 0.162690, 0.006713, -0.162987, -0.220998, 0.083108, 0.026168, -0.251240, 0.018553, -0.104916, -0.188408, -0.007697, -0.057978, -0.160972, -0.160025, -0.067211, -0.145218, -0.190131, 0.092764, 0.025449, -0.167894, -0.229953, 0.064689, 0.075397, -0.209588, 0.107188, 0.089073, -0.080405, 0.031624, 0.131544, -0.102374, 0.039610, 0.105508, -0.203861, 0.120127, 0.092031, 0.120020, 0.008069, -0.269261, 0.129556, -0.175342, 0.179533, 0.181329, -0.048755, -0.094702, -0.099701, -0.032849, -0.168873, 0.007508, -0.204996, -0.098034, 0.123244, -0.072101, -0.006969, -0.012494, 0.101649, -0.094537, 0.168231, -0.089403, -0.032065, 0.038520, -0.102243, 0.078368, -0.003533, 0.201117, 0.147341, 0.000962, 0.137667, -0.099660, 0.112765, 0.165554, -0.003054, -0.046399, 0.037375, -0.082632, -0.053002, 0.006530, -0.115165, -0.218031, 0.146812, -0.045703, -0.047095, -0.187636, -0.248226, 0.008975, -0.035089, -0.247149, 0.010909, -0.141086, 0.033582, 0.046870, 0.026986, -0.162250, 0.181453, -0.079880, -0.125142, 0.035112, -0.221431, -0.031269, -0.033955, -0.182166, -0.073946, 0.029919, -0.017677, 0.102744, 0.050007, 0.203223, -0.050583, -0.154773, 0.094398, 0.172041, -0.025008, -0.071187, -0.051416, -0.132822, -0.214228, -0.123545, 0.020750, 0.118510, -0.267256, -0.151250, -0.064021, 0.136177, 0.075619, -0.052630, -0.220219, 0.104414, -0.104515, 0.100698, 0.024376, 0.031545, -0.019857, 0.184470, -0.023951, 0.201691, -0.048933, -0.050628, -0.106438, -0.144221, 0.085044, -0.061666, -0.003440, 0.114548, -0.113571, -0.063113, -0.149883, -0.231086, 0.168807, 0.189000, -0.100231, -0.212070, 0.023967, -0.116457, -0.106547, 0.092277, -0.046945, 0.079230, -0.178069, -0.154461, -0.228762, -0.182785, -0.139319, 0.075915, 0.139459, -0.015411, -0.203283, 0.015147, 0.066272, -0.099117, -0.096452, 0.086900, -0.136055, 0.142824, -0.116338, 0.025016, -0.158700, 0.022083, 0.143109, -0.158336, 0.067653, 0.020425, 0.115204, 0.148361, -0.093780, 0.024555, 0.084137, -0.177413, 0.008700, 0.072282, -0.050387, 0.181537, 0.064798, 0.020360, -0.025410, -0.129684, 0.172169, 0.133576, -0.038328, -0.039753, -0.100537, -0.188232, -0.104797, 0.009509, -0.160821, -0.136193, 0.187715, 0.080495, 0.142507, -0.112630, 0.018149, -0.043601, -0.005145, 0.101457, 0.023155, -0.144749, -0.199948, -0.211947, -0.062993, -0.078606, 0.110997, -0.143283, 0.039227, 0.089242, -0.215382, 0.089589, 0.220947, 0.069715, -0.241524, -0.186060, 0.016640, -0.106317, -0.014027, -0.079524, 0.109182, 0.076188, -0.198620, -0.168251, -0.162477, 0.043841, -0.052630, -0.076567, -0.092701, 0.078072, 0.021543, 0.172751, 0.135313, 0.147821, 0.132467, -0.167929, -0.088592, 0.162098, -0.148587, 0.048029, -0.249911, 0.016675, 0.233101, -0.081811, 0.238881, 0.106396, 0.091837, -0.200439, -0.104207, -0.054120, 0.148718, -0.062928, -0.263816, -0.137687, 0.106893, 0.046282, 0.116825, 0.060096, -0.199340, -0.001481, -0.032136, 0.182016, -0.020477, 0.068802, 0.093807, -0.007107, 0.016390, -0.038848, -0.003995, -0.017074, 0.141418, 0.103226, -0.058193, -0.037460, -0.103801, -0.191240, 0.158296, -0.209071, 0.000973, 0.142015, -0.257622, -0.168149, -0.198492, 0.049495, 0.168498, -0.278393, 0.060121, -0.050809, 0.046848, 0.039852, 0.077347, 0.122856, -0.180872, 0.131647, -0.028642, 0.080471, 0.119349, 0.107144, 0.239806, -0.157665, -0.115875, -0.056992, 0.127495, 0.081902, -0.213950, 0.103815, -0.242172, -0.144274, 0.204785, 0.128645, -0.114874, 0.038003, 0.089306, 0.066272, -0.054892, -0.101228, 0.088170, 0.085930, -0.037906, 0.066707, -0.031384, -0.148178, -0.204148, -0.030258, -0.044266, 0.092554, -0.128923, 0.128254, -0.207565, -0.121365, 0.161021, 0.055441, 0.132810, -0.078076, -0.122189, 0.075973, 0.083530, 0.084315, -0.045538, 0.094101, -0.150394, 0.120926, 0.023058, 0.024018, 0.048490, -0.127737, -0.190660, 0.113682, 0.027284, -0.174501, 0.031990, 0.081054, -0.079009, -0.018344, -0.105399, 0.074602, -0.161182, 0.090526, 0.145769, -0.263158, 0.051536, -0.074488, -0.212269, -0.145064, 0.146161, -0.129024, -0.046608, -0.190778, -0.030772, -0.162515, 0.077865, -0.198759, -0.182206, 0.085732, -0.283933, -0.093270, 0.085093, 0.064581, 0.178087, 0.062132, -0.104943, -0.265024, 0.112701, 0.086531, -0.123810, -0.249047, -0.256520, 0.028357, -0.152399, -0.022150, -0.076901, -0.018218, -0.046563, -0.061145, -0.142526, -0.105981, -0.162923, -0.035189, -0.063013, 0.064950, 0.162953, -0.191534, -0.149038, 0.032344, -0.063380, -0.117506, -0.245808, 0.091629, -0.017261, -0.073465, -0.045410, 0.007090, 0.034745, 0.008076, -0.132518, -0.156898, -0.077817, 0.203200, 0.033604, -0.031922, 0.105459, -0.097677, 0.159753, -0.130119, -0.004635, 0.053019, -0.111458, -0.045096, 0.090431, -0.238046, -0.019331, -0.198789, -0.099207, -0.081391, -0.030734, -0.183423, 0.090616, 0.041235, 0.010797, -0.086633, -0.075456, -0.250842, -0.198288, 0.069771, -0.028523, -0.095769, -0.110560, 0.000893, 0.000040, -0.051924, -0.048272, -0.229717, 0.161767, -0.055050, -0.092417, 0.124414, 0.032945, -0.071673, -0.067353, -0.099497, -0.057776, -0.124306, 0.037371, 0.000361, -0.258351, -0.176557, 0.065653, 0.146299, -0.139200, -0.158257, 0.030842, -0.003725, -0.202649, 0.008102, -0.057356, 0.073134, 0.008535, -0.129729, -0.051063, -0.038931, -0.027468, -0.106782, -0.001024, -0.116288, -0.180409, -0.034534, -0.073670, 0.005906, 0.058219, 0.166522, -0.102660, -0.098151, -0.127832, -0.028517, -0.060918, -0.113861, -0.046391, 0.024097, -0.000475, -0.161964, -0.109885, -0.129191, 0.021787, 0.225193, 0.007721, 0.061646, -0.035113, -0.134712, 0.052947, -0.080252, -0.218266, 0.138702, -0.150738, 0.059385, 0.138550, 0.064942, -0.007138, -0.112035, 0.204377, -0.129377, -0.021014, 0.149506, -0.001235, -0.077465, -0.160133, -0.117720, 0.092737, -0.029005, 0.174047, -0.274779, -0.250030, 0.078172, -0.090331, 0.042961, -0.205316, 0.046367, -0.056894, -0.173929, 0.076132, -0.147334, -0.039802, -0.266360, -0.284472, -0.015277, -0.217796, 0.034299, 0.030395, 0.000070, -0.014245, -0.205233, 0.016903, -0.048655, -0.151058, 0.114937, 0.057784, 0.038171, -0.219878, 0.079477, 0.097282, -0.021168, -0.081827, 0.088759, -0.058871, 0.070619, -0.205786, -0.067125, 0.106157, -0.062420, -0.136652, -0.180082, -0.065296, -0.286946, -0.321869, 0.017554, 0.089872, -0.105208, 0.044293, 0.248013, -0.173252, -0.109481, 0.202816, -0.014991, 0.124017, -0.067284, -0.023998, 0.088478, 0.101868, 0.081817, 0.209412, -0.018781, -0.172477, -0.164562, 0.200007, 0.056884, 0.106272, -0.182880, -0.123781, 0.063267, -0.230638, -0.019055, -0.205419, 0.197541, -0.198720, -0.182181, 0.110510, -0.084713, 0.065407, -0.049739, 0.156435, -0.224698, 0.094290, 0.014365, -0.190435, 0.126705, -0.059463, 0.057626, 0.069520, -0.047589, -0.157757, 0.138826, 0.176764, -0.288364, -0.024494, -0.205077, 0.019677, -0.138235, 0.125638, 0.014956, -0.232807, -0.061307, 0.082854, -0.175044, 0.031433, -0.183093, 0.093276, 0.027900, -0.209902, 0.159516, 0.129424, 0.132976, 0.040934, 0.128310, -0.115805, 0.160791, 0.200437, 0.120027, -0.169269, 0.001254, -0.122004, -0.111766, -0.116197, 0.107472, 0.124729, -0.004954, -0.095255, 0.073652, 0.004850, -0.178254, 0.195797, -0.031146, -0.259319, -0.115599, -0.063144, -0.061969, 0.149608, -0.014443, -0.213948, 0.008068, 0.144077, -0.143199, -0.070661, -0.090459, 0.122777, -0.055731, 0.107613, -0.023732, 0.020959, 0.093576, -0.187325, 0.074573, 0.007694, 0.117199, 0.041512, -0.216200, -0.130893, -0.149750, 0.028815, -0.030344, -0.116414, -0.317162, -0.040079, 0.242659, -0.023888, -0.066037, 0.052766, -0.005770, 0.050451, -0.208458, 0.191133, -0.078927, -0.090132, -0.181439, 0.017455, -0.037453, -0.011490, -0.059334, -0.032730, -0.006085, -0.063982, -0.026299, 0.109608, -0.084109, -0.012514, -0.013087, -0.065923, 0.004334, 0.010522, -0.033329, -0.109663, 0.254545, 0.172810, -0.163591, 0.120675, -0.145430, 0.151358, -0.078560, -0.037670, -0.154208, 0.069605, -0.067404, -0.119043, 0.032602, 0.079160, 0.016203, -0.089354, -0.060417, -0.162385, -0.212389, -0.221961, 0.068451, -0.107366, -0.121543, -0.101876, 0.016305, 0.125544, -0.033034, -0.040435, -0.076167, 0.195144, 0.068947, -0.065570, -0.105697, -0.124721, -0.109227, -0.083588, 0.099832, 0.003592, -0.160067, 0.003259, 0.041199, -0.083822, -0.132558, -0.256203, -0.182740, 0.001317, -0.137657, -0.082421, 0.046106, 0.120890, 0.025548, -0.126929, 0.107434, 0.019413, 0.090971, -0.067734, 0.123079, 0.127130, -0.161999, -0.005005, 0.048149, -0.023897, -0.270545, -0.111089, 0.004118, 0.033362, -0.027953, 0.054008, 0.152816, -0.201762, 0.021524, -0.123197, -0.073559, 0.000524, -0.091507, -0.106242, 0.050329, -0.108801, -0.101153, -0.064999, -0.002875, 0.039322, -0.107689, -0.154053, -0.202276, -0.040283, 0.089812, 0.114359, -0.107079, -0.124529, -0.001914, -0.104789, -0.121565, -0.198390, -0.099632, -0.006911, -0.045216, -0.029867, 0.030992, -0.083115, -0.039788, 0.017990, 0.004738, -0.146365, 0.212923, 0.018532, -0.198817, -0.014912, -0.021895, 0.056025, 0.134704, 0.052262, 0.077839, -0.074575, -0.030728, 0.051926, -0.134101, -0.065329, 0.095441, 0.005362, -0.320066, -0.031660, 0.185336, -0.185066, -0.244708, -0.041238, -0.240934, 0.289305, 0.085717, 0.070756, -0.281231, -0.121665, 0.017694, 0.043168, 0.018245, 0.117926, -0.134891, 0.173788, -0.016483, 0.074033, 0.297291, -0.077766, -0.096016, -0.143047, 0.054483, -0.159745, -0.015035, -0.079806, -0.192738, -0.229282, -0.033435, -0.210121, -0.120133, 0.081383, 0.028186, -0.233440, -0.005699, -0.141221, 0.161547, 0.060737, -0.041088, -0.145830, 0.006742, -0.148999, 0.135203, 0.102135, -0.238380, 0.122228, 0.041691, -0.162923, -0.041621, 0.034483, -0.072151, -0.106803, -0.070408, -0.161970, 0.014867, 0.027113, -0.124863, -0.136033, -0.094630, -0.129611, 0.053116, 0.009706, -0.195417, -0.151510, -0.067206, 0.139619, 0.139601, 0.034085, 0.056369, 0.079887, -0.058680, 0.139363, -0.165965, -0.116522, -0.065965, 0.161519, -0.058847, 0.010203, -0.180771, -0.010577, -0.093030, 0.129600, 0.164807, -0.038184, -0.152913, -0.150552, -0.034221, -0.080638, -0.145570, -0.164487, -0.153948, -0.123227, -0.136960, -0.182059, -0.143404, -0.190808, -0.041683, -0.101558, -0.205040, 0.106900, -0.119287, 0.062814, -0.006110, -0.051024, -0.154184, -0.103544, -0.112718, -0.038922, 0.215685, -0.091556, 0.110361, -0.118157, -0.128787, 0.085860, -0.296992, 0.088935, -0.117518, 0.076616, -0.241626, -0.151477, 0.257687, -0.197329, -0.074681, -0.111951, 0.084828, -0.143288, 0.031309, -0.118217, -0.294245, -0.193350, -0.042170, -0.051293, -0.056437, -0.097944, -0.068279, -0.082731, -0.115753, 0.102119, 0.128756, -0.128144, 0.023206, 0.053891, -0.317280, -0.090716, -0.048617, -0.201192, 0.030243, 0.006836, 0.008797, 0.170371, -0.113556, -0.150117, -0.184408, -0.039981, 0.085722, -0.163927, -0.088385, -0.135078, 0.120191, -0.026627, -0.042047, 0.050042, 0.131262, 0.035964, 0.166282, -0.128620, -0.198723, -0.217690, -0.040826, 0.102168, -0.020908, -0.013998, -0.224456, -0.218090, -0.147928, 0.118010, 0.106042, -0.028700, 0.235288, -0.180627, -0.198808, -0.249863, -0.064488, 0.017811, 0.166005, -0.213845, 0.138073, -0.153009, 0.141843, -0.051419, -0.075694, -0.226131, -0.041074, -0.207081, 0.040820, -0.064222, -0.028781, 0.168728, 0.101631, -0.161025, 0.093556, -0.202608, 0.108386, -0.153070, 0.192274, -0.145241, -0.000211, 0.236275, -0.087635, -0.151944, -0.028237, 0.198736, -0.024313, -0.087090, -0.097063, -0.121538, -0.099224, 0.134001, -0.174923, 0.151579, -0.053231, -0.247944, -0.088981, -0.211388, -0.063122, -0.018182, 0.168559, -0.169690, -0.055651, 0.025104, 0.185304, -0.144953, -0.049440, 0.119042, -0.046729, -0.055920, 0.180785, -0.090310, 0.157958, -0.117315, 0.043618, -0.134080, 0.056683, -0.077463, -0.241500, 0.129426, -0.142416, 0.023727, 0.108929, -0.008048, 0.172686, -0.132356, -0.196406, -0.184002, 0.210628, -0.238060, -0.089066, 0.114596, 0.153111, 0.194562, 0.161066, -0.035873, 0.036367, -0.155359, 0.100467, -0.026104, 0.356755, -0.082889, 0.026330, -0.048655, -0.118040, 0.029410, -0.169095, 0.000227, 0.103414, 0.181038, -0.095122, -0.093822, 0.081849, -0.091800, 0.081307, 0.068839, -0.082793, -0.111909, 0.114605, 0.013529, 0.014640, -0.110074, 0.100217, -0.050205, 0.122569, -0.025452, -0.140571, -0.102917, -0.259463, -0.041072, 0.286599, -0.108083, 0.061381, 0.046828, -0.140044, 0.062607, 0.055307, -0.086436, -0.228696, 0.050932, 0.117816, 0.102888, -0.166034, 0.226874, 0.022948, -0.109273, -0.160216, 0.047745, 0.172978, 0.058415, -0.126457, -0.043911, 0.017664, 0.007508, 0.072441, 0.103484, 0.085472, 0.019245, -0.137672, 0.061656, 0.124268, -0.181649, -0.003858, 0.013738, 0.008420, 0.043954, 0.048462, -0.140401, -0.031369, 0.051175, -0.147290, -0.226342, -0.100782, -0.147707, 0.129768, 0.119781, -0.055445, -0.100545, -0.073053, 0.085573, -0.074556, -0.105671, -0.036404, -0.072882, 0.075968, 0.063639, -0.194386, -0.122092, -0.002620, -0.022566, -0.133343, 0.162517, 0.050876, -0.199029, 0.188501, 0.167689, -0.071162, 0.118603, 0.109654, -0.110553, 0.138290, 0.142590, -0.102962, 0.045384, 0.012512, -0.102174, -0.140773, -0.094162, 0.010323, 0.155468, -0.142019, -0.097794, -0.137002, -0.212146, 0.207217, -0.017213, 0.002942, 0.034605, 0.107504, 0.150266, -0.129505, 0.192782, -0.028705, -0.202198, -0.147815, -0.153301, 0.174837, 0.060969, 0.128735, 0.105888, 0.073072, 0.088999, -0.002995, -0.193849, -0.173289, 0.083937, -0.146552, 0.142054, -0.139680, -0.000768, -0.076366, -0.059695, 0.032080, -0.010387, 0.051921, -0.102333, -0.071009, 0.175738, -0.134685, -0.134976, -0.095431, 0.205827, -0.073887, 0.094985, -0.191911, 0.164504, -0.086110, -0.108445, 0.061845, 0.162021, 0.028200, 0.119438, -0.245631, 0.091793, 0.114317, -0.021548, 0.107032, 0.038590, 0.093562, -0.205856, 0.118910, -0.084905, 0.021004, -0.198377, -0.234301, -0.211129, 0.070893, 0.022674, -0.051338, 0.153045, -0.149085, -0.122123, 0.079959, -0.204106, -0.200147, 0.090186, 0.084070, 0.131274, -0.088271, 0.169127, -0.101847, 0.176898, 0.156308, 0.027733, 0.075918, -0.044774, -0.035376, 0.027992, 0.050958, -0.174579, 0.092923, -0.093785, -0.139114, -0.086600, -0.116225, 0.079024, -0.074963, -0.027205, 0.063837, -0.077457, 0.097615, -0.170624, -0.204657, -0.174123, 0.252476, -0.037762, -0.003866, -0.066153, 0.032779, -0.063880, 0.102435, -0.165147, 0.003097, -0.019100, 0.193608, 0.024472, 0.017538, 0.040808, -0.101324, -0.124583, -0.220176, -0.176091, -0.236821, 0.080546, -0.147749, -0.021607, -0.064803, -0.108025, 0.158381, 0.062731, -0.012334, -0.053412, -0.167796, -0.192720, -0.003843, 0.094745, -0.155300, 0.099702, -0.084310, -0.010902, 0.030403, -0.033079, 0.012516, -0.123602, -0.057762, 0.091336, -0.052454, 0.047064, 0.102744, 0.021584, -0.068199, -0.177980, -0.174477, 0.108816, 0.072409, -0.097811, 0.006908, 0.109265, 0.069252, 0.082388, -0.013773, 0.083408, -0.123182, 0.143093, -0.027379, 0.216197, 0.204592, -0.202415, -0.173952, -0.049781, -0.209224, 0.207557, -0.108861, 0.012178, -0.180074, -0.204747, 0.012663, -0.117213, -0.078747, -0.232379, -0.082473, 0.222548, -0.076128, 0.017688, 0.185962, 0.059833, 0.070901, 0.145850, 0.166014, -0.001596, 0.174953, 0.097180, -0.047201, 0.140861, -0.002166, -0.015422, 0.082614, 0.018298, -0.158532, -0.081273, 0.026782, 0.010039, 0.014152, -0.113708, 0.021807, -0.006415, 0.134055, -0.024455, 0.166605, 0.119609, -0.240276, 0.011147, -0.070938, -0.001916, -0.190984, -0.020498, 0.049692, 0.119988, 0.012101, -0.079877, 0.104347, 0.115889, -0.000701, -0.000200, -0.116832, -0.053406, 0.127320, 0.123170, -0.223954, 0.077958, 0.000277, 0.190590, 0.119747, 0.106785, 0.065563, 0.016657, -0.069956, -0.145500, -0.127351, -0.048157, -0.251979, 0.125064, -0.110993, 0.078520, -0.005572, -0.201606, 0.109670, -0.176686, 0.156523, 0.133993, -0.091991, 0.168931, -0.148177, -0.050699, -0.120765, -0.139533, 0.058259, 0.140237, 0.092177, -0.165459, -0.171207, 0.156731, 0.010243, -0.049143, -0.198165, 0.058386, -0.002632, -0.010948, -0.065568, -0.082094, 0.111951, -0.213757, -0.177344, 0.045442, 0.009229, -0.081340, -0.063801, 0.186457, 0.136439, -0.109015, 0.086114, 0.111018, -0.081917, -0.077104, -0.197834, -0.215515, 0.045228, -0.149443, -0.175919, 0.159206, -0.214795, 0.049048, -0.150895, 0.177309, -0.133976, -0.049341, -0.101059, -0.035851, -0.128504, 0.057545, 0.148281, -0.165562, 0.097207, 0.138636, -0.172084, -0.049035, -0.149735, 0.085481, -0.005862, 0.022614, -0.301166, 0.073367, 0.035003, -0.048621, 0.069253, 0.041897, -0.004374, 0.075960, -0.060290, 0.138160, 0.120225, 0.085650, -0.208537, 0.096014, 0.044026, 0.042850, 0.103294, 0.101432, 0.030810, -0.296734, -0.137424, 0.143252, 0.145805, -0.086185, 0.120815, -0.035621, 0.022993, 0.133212, -0.172715, 0.113733, -0.170444, -0.036648, 0.122507, -0.022651, 0.110245, 0.164986, -0.102638, -0.163859, -0.129321, 0.024643, -0.008650, 0.003262, 0.188762, -0.044951, -0.100630, 0.129388, 0.057905, 0.111092, 0.097379, 0.180758, -0.122092, -0.061474, 0.097122, -0.016703, -0.092755, -0.217754, -0.209254, 0.169666, -0.168835, 0.120574, -0.075259, -0.146628, 0.023180, -0.181881, -0.070199, 0.201167, -0.086352, -0.033172, 0.029317, -0.147238, -0.169502, 0.026048, -0.126043, -0.150882, -0.246272, -0.086376, 0.114050, -0.037291, -0.077498, 0.131446, 0.134411, -0.065761, 0.052115, -0.103191, 0.036951, -0.105550, -0.174234, -0.113685, 0.169620, -0.111003, -0.190180, -0.070703, -0.011564, 0.170409, -0.213383, -0.093098, -0.001624, 0.128783, 0.108914, -0.304261, -0.043003, 0.030753, 0.004043, -0.094789, 0.165093, 0.031420, 0.103349, 0.053297, -0.224531, -0.036606, 0.016023, -0.229925, 0.018866, -0.094369, -0.004789, -0.117526, -0.017096, 0.166951, 0.041755, -0.016534, 0.032813, -0.079353, -0.091808, -0.141489, 0.000641, 0.014971, -0.044141, -0.172049, -0.077523, 0.106444, -0.053978, -0.140208, -0.167674, -0.057589, 0.031635, 0.051585, 0.228365, -0.278278, 0.005538, -0.040600, -0.008821, -0.229175, -0.150135, -0.048334, -0.063206, -0.176003, 0.017721, 0.280622, 0.036771, 0.028169, 0.035114, 0.173123, 0.015005, 0.026818, 0.013097, 0.174614, -0.055922, 0.049859, -0.079898, -0.094391, -0.148679, 0.104692, 0.092321, -0.096423, 0.169699, 0.076722, -0.191469, -0.095258, -0.112098, -0.109355, -0.155259, 0.060463, 0.039525, -0.048619, -0.098098, -0.039907, -0.006702, -0.148284, -0.126526, 0.021500, -0.052005, -0.143786, 0.104853, -0.211339, 0.014862, -0.028785, -0.077053, -0.218324, 0.112712, -0.070995, -0.094271, -0.060391, -0.202425, 0.002345, -0.030716, -0.146052, 0.001556, -0.164822, 0.037714, -0.072036, -0.161283, -0.130253, 0.057649, -0.001839, 0.047250, -0.058188, 0.014529, -0.228346, 0.225228, -0.023914, 0.133087, 0.086785, -0.038637, 0.056942, -0.125695, 0.081435, -0.067135, 0.205670, 0.027072, -0.091504, -0.204132, 0.043087, 0.082807, -0.095363, 0.184644, -0.216296, 0.080196, -0.061449, 0.048607, -0.191740, -0.084450, -0.225042, -0.136752, -0.167331, -0.001254, -0.101233, -0.008365, 0.126993, -0.073219, -0.113536, 0.073879, -0.098733, 0.172418, -0.198177, 0.192814, -0.122041, -0.060191, -0.014931, 0.163615, 0.067764, -0.245190, 0.178596, -0.136161, -0.044688, -0.142136, 0.182072, 0.069366, 0.028530, -0.070855, -0.174058, -0.020019, 0.118313, 0.147296, 0.010455, -0.009949, -0.016825, -0.202637, -0.092267, 0.178319, 0.056175, -0.129320, 0.100304, -0.182421, -0.058295, 0.101226, -0.040390, -0.163760, 0.140207, -0.183046, -0.084880, 0.045066, -0.133398, -0.018702, -0.007750, 0.182355, 0.032732, 0.052878, -0.055891, -0.242827, -0.185519, -0.177503, -0.027939, 0.044171, 0.150245, -0.014234, 0.112920, -0.138517, 0.026886, 0.002449, -0.065427, 0.118718, -0.156467, 0.016188, 0.045635, -0.073365, -0.104475, -0.000712, 0.089148, 0.064683, -0.087668, 0.072877, -0.062352, 0.164486, -0.179810, 0.150326, 0.034267, 0.083289, -0.135315, -0.078507, 0.114422, -0.139795, 0.072093, 0.045491, 0.071670, -0.095322, -0.025386, 0.045614, -0.045319, 0.027453, -0.017968, 0.054306, -0.045315, -0.133014, 0.025252, 0.038265, -0.142094, -0.252877, -0.093276, 0.158396, -0.059512, 0.081310, -0.103027, -0.210447, -0.021172, 0.105464, -0.214733, -0.136482, -0.141165, -0.123488, 0.163751, 0.037223, -0.002330, -0.041271, 0.105434, -0.089937, -0.132007, -0.014517, -0.178780, 0.066776, 0.012766, -0.118609, -0.011695, 0.154159, 0.144913, -0.223193, -0.153674, -0.140621, -0.156612, -0.074044, 0.027742, 0.123790, 0.085903, 0.024382, -0.214596, 0.014919, -0.081420, 0.184341, 0.115362, 0.059852, -0.210994, 0.118274, -0.188437, -0.016531, -0.061721, -0.270835, -0.077802, -0.125344, -0.052194, -0.179581, -0.190326, -0.079306, 0.020550, -0.051439, -0.121190, 0.088697, -0.016546, -0.036693, 0.090806, -0.190309, 0.038711, 0.054625, 0.094326, 0.099890, -0.125696, 0.050182, 0.067814, -0.113649, 0.051156, -0.119833, -0.049884, 0.020490, -0.090113, -0.132251, -0.135071, 0.179905, -0.041647, -0.108981, 0.079675, -0.038361, 0.111527, -0.258289, -0.030221, -0.128926, 0.019172, -0.177219, -0.007955, -0.178778, 0.127273, 0.065075, 0.177154, -0.217254, -0.126796, 0.126726, -0.111803, -0.032864, -0.137408, -0.080912, -0.209764, -0.067656, -0.137620, -0.064496, -0.020262, -0.006527, -0.054540, -0.063401, -0.072403, -0.137469, 0.068536, -0.138401, -0.161253, -0.162836, -0.104828, 0.095207, 0.077288, -0.305322, 0.085743, -0.018109, 0.152192, -0.185967, -0.223404, -0.162980, -0.006216, -0.090014, -0.304059, -0.040610, -0.161808, -0.106053, 0.069236, -0.124966, -0.079949, 0.130094, -0.012569, -0.247941, -0.311043, 0.076641, -0.254534, 0.168732, 0.151197, 0.096066, -0.109540, -0.133976, 0.020003, 0.071978, -0.115032, 0.000622, 0.078090, -0.051392, -0.076593, 0.027368, 0.156209, -0.008914, 0.058649, -0.183826, 0.037149, 0.049349, -0.197463, 0.062533, 0.213416, -0.053868, -0.064938, -0.203398, 0.139220, -0.057218, -0.353997, -0.208465, -0.035827, -0.167311, -0.273190, 0.026726, -0.101909, 0.077252, -0.155960, 0.169625, -0.100422, 0.011970, 0.049087, 0.130031, -0.291059, -0.193894, 0.097732, 0.161230, 0.140426, -0.220959, 0.015363, -0.256408, 0.059064, -0.138914, -0.076260, 0.035331, -0.065078, -0.208651, -0.161200, 0.000114, -0.025323, -0.200176, -0.061118, 0.171024, 0.091732, -0.132836, 0.199614, -0.028562, 0.008729, -0.246628, 0.049238, 0.146236, 0.133155, -0.015795, -0.176688, -0.020591, 0.061433, 0.040517, 0.002126, -0.065077, 0.122625, 0.004215, -0.115735, 0.130443, 0.024980, -0.191152, 0.044253, -0.119547, 0.166143, 0.158529, -0.135224, 0.137646, -0.022944, -0.092697, -0.110082, 0.055043, 0.087793, -0.217556, -0.124660, -0.024366, -0.037417, -0.041360, 0.207956, -0.204809, -0.099651, -0.064103, 0.018620, -0.036742, -0.082300, -0.046805, 0.085820, 0.005664, -0.097973, 0.025471, 0.151985, 0.152762, -0.068417, 0.132164, 0.024411, 0.163285, -0.150605, 0.115086, -0.103740, -0.137768, -0.052945, -0.175771, 0.060126, 0.087909, -0.040286, -0.187278, 0.099051, 0.052965, 0.173914, -0.028730, 0.064500, -0.114007, 0.164003, -0.079744, -0.112161, 0.057059, 0.005838, -0.140348, -0.247910, -0.065861, -0.131887, -0.024241, 0.043749, -0.000074, 0.110206, -0.196882, -0.053262, -0.200684, -0.030804, -0.054183, -0.113677, -0.054359, 0.092339, -0.106815, -0.008589, -0.124783, 0.035536, 0.062986, 0.108620, 0.143586, 0.148991, -0.186290, -0.264083, 0.134763, -0.267610, 0.039798, -0.294081, 0.048332, 0.009111, -0.148995, 0.049602, -0.252272, 0.028599, -0.202086, 0.153768, -0.236532, -0.171448, 0.162534, 0.064755, 0.056175, 0.022952, 0.250896, -0.029718, -0.173681, 0.158051, 0.040543, -0.231278, 0.007338, -0.146466, -0.048713, 0.098086, -0.142327, 0.136999, -0.108787, 0.121871, 0.063656, 0.009787, 0.020407, 0.102134, -0.083000, 0.010565, -0.048279, -0.176006, 0.192838, -0.191778, -0.011151, -0.034629, -0.137959, -0.156114, -0.208282, -0.111760, -0.153745, 0.046481, -0.014690, -0.074393, 0.131933, 0.139451, -0.055038, -0.018948, 0.081301, 0.054266, -0.207600, -0.132152, -0.085538, 0.110824, 0.006603, -0.044691, 0.100401, 0.057999, -0.123625, -0.123461, 0.156083, 0.015191, -0.065772, -0.142643, -0.092887, 0.134659, 0.142926, -0.146464, 0.146968, 0.056252, -0.092639, -0.132505, -0.218644, -0.062490, -0.113292, 0.031208, -0.137225, -0.102919, -0.236363, 0.133594, 0.048363, -0.024879, -0.078548, -0.141144, 0.101765, -0.140912, 0.069862, 0.150613, 0.072240, 0.165092, -0.236113, -0.191374, -0.101077, 0.108025, 0.166719, -0.238632, 0.152048, -0.052795, 0.150607, 0.055162, 0.012433, -0.066308, -0.011505, -0.185655, 0.151592, -0.107767, 0.026636, -0.003549, 0.147447, 0.050168, -0.024285, 0.131619, 0.168610, -0.072330, -0.028232, 0.128439, 0.099897, 0.023590, -0.066392, -0.201158, 0.078802, 0.094906, -0.000663, 0.071690, 0.134810, -0.007040, 0.014827, -0.197253, -0.009845, 0.035017, 0.132641, -0.121228, 0.134291, 0.117331, -0.188520, -0.152289, -0.141274, -0.038179, -0.100922, -0.112152, 0.136913, -0.262308, 0.016783, 0.253381, 0.038586, -0.153809, -0.178875, -0.015969, -0.153369, -0.015771, 0.033027, -0.072162, -0.057355, -0.077830, -0.045508, -0.075716, -0.288942, 0.088621, -0.100052, -0.088039, -0.105165, -0.018854, 0.073136, 0.179621, -0.145362, -0.167369, -0.095839, -0.179292, -0.140104, 0.013484, -0.145016, -0.090266, -0.059632, -0.040548, 0.173645, 0.126563, 0.024837, 0.140913, 0.066702, -0.038213, 0.041581, -0.061723, -0.197405, 0.127345, 0.123313, 0.035559, 0.078090, -0.289412, -0.203056, -0.129500, 0.104932, -0.135210, -0.219854, 0.161049, -0.059190, -0.060268, 0.027543, -0.051009, -0.191298, 0.042308, 0.019076, -0.168354, 0.041126, -0.005694, -0.071274, -0.138837, -0.134504, -0.118111, 0.011635, -0.106810, -0.196882, 0.118571, -0.118696, -0.039983, 0.090979, 0.039514, -0.182780, 0.102375, -0.003887, -0.076427, -0.035515, 0.040621, 0.140793, -0.002671, -0.169209, -0.026444, 0.078911, -0.082160, 0.150896, -0.052593, -0.031593, -0.057499, 0.143073, 0.099486, 0.159700, 0.016986, 0.015134, -0.132928, -0.068091, -0.130855, -0.116659, 0.005557, -0.183294, -0.105724, 0.102137, -0.199357, -0.043928, -0.048290, 0.049384, -0.074718, 0.130312, 0.014877, 0.086195, 0.039925, 0.192903, -0.009462, 0.083391, -0.083780, -0.107732, -0.078282, 0.041608, 0.148125, -0.108374, 0.034591, -0.138861, 0.086235, -0.107254, 0.042563, -0.015521, 0.083286, 0.127555, 0.100179, -0.057363, -0.107776, -0.045854, -0.150989, -0.027542, -0.010367, 0.057750, 0.169215, 0.194196, 0.105961, 0.015154, -0.079443, 0.184819, -0.012438, -0.104517, 0.097260, 0.045942, -0.087822, 0.102265, 0.039257, -0.209432, -0.023566, -0.177704, -0.027071, -0.174235, 0.069330, -0.181450, 0.100489, -0.051742, -0.055866, -0.172310, -0.129962, 0.051289, -0.075422, -0.050917, -0.058220, -0.009143, 0.057268, -0.150454, -0.097749, 0.018910, -0.051320, 0.031283, -0.283164, 0.142133, -0.238375, -0.160468, 0.003632, -0.068129, -0.031635, 0.050023, 0.137219, -0.133289, 0.184128, 0.030182, -0.012697, -0.115159, -0.015287, -0.178916, -0.209030, -0.110985, 0.159423, 0.043565, 0.066585, -0.207925, -0.247766, -0.022268, -0.253016, -0.185516, -0.012988, 0.096451, 0.005457, -0.232635, -0.212538, 0.047166, -0.024269, -0.098210, -0.119028, -0.052694, -0.039378, 0.090767, 0.261124, 0.092100, -0.030561, -0.185455, -0.166724, -0.230407, -0.141056, -0.129484, -0.107713, 0.147920, -0.136659, 0.192888, -0.005773, -0.124367, -0.236723, 0.131806, -0.109306, 0.044002, -0.174655, 0.043329, -0.068857, 0.032437, 0.024313, -0.134711];
    bias_1 : ARRAY[0..59] OF REAL := [0.366822, 0.481196, -0.074898, -0.790819, -0.115352, 1.205088, -0.153314, -0.030682, 0.937615, 0.445205, -0.117856, -0.930737, 0.281899, -0.016763, -0.230018, -0.118161, 0.151101, 0.102791, 0.697760, 0.898044, 0.066976, 1.419901, -0.109749, -0.780416, 0.623116, 1.375208, -1.140123, -0.095345, -0.891303, 1.191562, -0.046032, -0.347076, -0.367348, -0.247266, 1.030839, -0.077343, 0.185900, -0.138577, 1.299610, -0.057316, -0.070718, 0.017384, 0.138374, 1.025729, -0.059147, -0.122236, -0.114517, 0.144933, 0.942493, 0.001337, 0.909855, -1.173982, -0.783042, -0.359816, -0.232239, 0.094986, -0.266255, -0.458538, -0.115432, 0.084889];

    weights_2 : ARRAY[0..179] OF REAL := [-0.361096, -0.212831, -0.207744, 0.143652, -0.318005, -0.242553, -0.203271, 0.222259, -0.198057, -0.068261, -0.208135, -0.019708, 0.044099, 0.144559, 0.255032, 0.340644, 0.082924, 0.272515, -0.014006, -0.230609, -0.027759, -0.238744, 0.101299, -0.243001, 0.235500, -0.034529, -0.270894, 0.177581, 0.053919, -0.152719, -0.002021, -0.047382, 0.107008, -0.143225, -0.318478, -0.164218, 0.148955, -0.157341, 0.128601, 0.020439, 0.165380, 0.162863, 0.115839, -0.196290, 0.014463, -0.130199, 0.040108, 0.094993, 0.134977, -0.065247, 0.156363, 0.167069, 0.120219, -0.189792, -0.270223, 0.140174, 0.032212, 0.073417, -0.006858, -0.191435, 0.188309, 0.206222, -0.016329, 0.105434, 0.192674, -0.211180, 0.086663, 0.209301, 0.284761, 0.070211, -0.055109, 0.135917, -0.059921, 0.179572, 0.086714, -0.131614, -0.188568, -0.274244, 0.268252, 0.034215, 0.201453, 0.003005, 0.181906, 0.289455, 0.291069, -0.006117, 0.227284, 0.214860, -0.020120, -0.073110, -0.113842, 0.009435, 0.036648, 0.082109, -0.020422, 0.225021, -0.173540, -0.096475, -0.025091, 0.069112, 0.135963, 0.159734, 0.283007, -0.265928, 0.215183, -0.268602, 0.212231, -0.216117, -0.204204, -0.288449, -0.179859, -0.177738, -0.021980, 0.012611, 0.182575, -0.266667, 0.034078, -0.126150, 0.021102, 0.069167, -0.288389, -0.123025, -0.200112, 0.116275, 0.036289, -0.147439, 0.090122, 0.066952, -0.039597, 0.156977, -0.133114, -0.070397, -0.124950, 0.163808, -0.257259, -0.129965, 0.028123, -0.150497, 0.016644, -0.046663, 0.059387, -0.030999, -0.061351, -0.070851, -0.129827, -0.174570, -0.192345, -0.204283, 0.110348, 0.167108, 0.350771, -0.301933, -0.197836, 0.310112, 0.003010, 0.241587, -0.040090, -0.133023, 0.027663, 0.104344, 0.068014, 0.176260, -0.064415, -0.119342, -0.064906, -0.071797, 0.175540, 0.115916, 0.005464, -0.065432, 0.180886, -0.022479, -0.048810, 0.070312, 0.027939, 0.118338, -0.214642, -0.033401, 0.091202, 0.147469];
    bias_2 : ARRAY[0..2] OF REAL := [-0.040190, 1.222343, -1.097594];

END_VAR

VAR
    (* Buffer allocation variables *)
    buffer_0 : ARRAY[0..59] OF REAL;
    buffer_1 : ARRAY[0..79] OF REAL;

    (* Temporary computation variables *)
    i : DINT;
    j : DINT;
    sum : REAL;
    max_val : REAL;
    exp_sum : REAL;

END_VAR

(* Layer 0: Fused Linear + RELU *)
FOR j := 0 TO 79 DO
    sum := 0.0;
    FOR i := 0 TO 4 DO
        sum := sum + input_data[i] * weights_0[i * 80 + j];
    END_FOR;
    buffer_1[j] := MAX(sum + bias_0[j], 0.0);
END_FOR;

(* Layer 1: Fused Linear + RELU *)
FOR j := 0 TO 59 DO
    sum := 0.0;
    FOR i := 0 TO 79 DO
        sum := sum + buffer_1[i] * weights_1[i * 60 + j];
    END_FOR;
    buffer_0[j] := MAX(sum + bias_1[j], 0.0);
END_FOR;

(* Layer 2: Fused Linear + SOFTMAX *)
FOR j := 0 TO 2 DO
    sum := 0.0;
    FOR i := 0 TO 59 DO
        sum := sum + buffer_0[i] * weights_2[i * 3 + j];
    END_FOR;
    output_data[j] := sum + bias_2[j];
END_FOR;

max_val := output_data[0];
FOR i := 1 TO 2 DO
    IF output_data[i] > max_val THEN
        max_val := output_data[i];
    END_IF;
END_FOR;

exp_sum := 0.0;
FOR i := 0 TO 2 DO
    output_data[i] := EXP(output_data[i] - max_val);
    exp_sum := exp_sum + output_data[i];
END_FOR;

FOR i := 0 TO 2 DO
    output_data[i] := output_data[i] / exp_sum;
END_FOR;

END_FUNCTION_BLOCK

(* ---- test8_1k.st ---- *)
FUNCTION_BLOCK NeuralNetworkFB

VAR_INPUT
    input_data : ARRAY[0..4] OF REAL;
END_VAR

VAR_OUTPUT
    output_data : ARRAY[0..2] OF REAL;
END_VAR

VAR CONSTANT
    weights_0 : ARRAY[0..39] OF REAL := [-0.044422, 0.480684, -0.074478, 0.030278, -0.049364, 0.445707, -0.186376, 0.244870, 0.104984, -0.315322, -0.217575, -0.258209, -0.076724, -0.470795, -0.092567, -0.403755, -0.254578, -0.556995, -0.307716, 0.411375, -0.015841, -0.067324, 0.335760, 0.370447, -0.002549, -0.080746, -0.408668, 0.444774, 0.189295, -0.154797, -0.098240, -0.107421, 0.586036, -0.265400, 0.323485, 0.458571, 0.512554, -0.201372, 0.445545, -0.377168];
    bias_0 : ARRAY[0..7] OF REAL := [-2.043351, -0.191602, -0.271955, -1.295284, -0.525869, -0.436923, -1.763881, 0.086360];

    weights_1 : ARRAY[0..63] OF REAL := [0.214678, 0.073610, 0.399105, 0.565031, 0.372911, 0.203032, 0.186051, 0.165617, -0.031932, 0.032175, -0.507027, -0.545832, -0.132381, -0.185731, -0.476689, -0.572535, -0.075155, -0.096659, -0.030058, 0.133983, -0.124660, -0.413428, -0.220973, -0.287707, -0.080595, 0.092690, -0.455686, 0.113307, -0.245535, 0.252006, -0.565568, -0.484327, 0.140556, 0.394913, -0.515051, -0.199015, -0.554787, 0.016071, -0.058181, 0.418473, 0.030105, -0.205639, 0.029723, -0.547427, -0.129825, 0.161570, 0.131558, -0.272732, 0.627360, -0.063176, -0.465176, 0.237206, -0.336560, 0.488126, 0.434088, -0.219548, -0.202927, -0.239346, 0.211005, -0.218231, 0.130038, -0.834673, -0.318850, 0.078278];
    bias_1 : ARRAY[0..7] OF REAL := [-0.213226, -0.920354, 0.001473, -1.331399, -0.396995, -0.915665, -0.540294, -0.404236];

    weights_2 : ARRAY[0..63] OF REAL := [0.255640, 0.491090, -0.279060, -0.321454, 0.173054, -0.324807, 0.056291, -0.142179, 0.366396, -0.073566, -0.005377, -0.527611, 0.408393, -0.187448, -0.151590, 0.581381, -0.292516, 0.122751, 0.231838, 0.288276, 0.019622, -0.399430, -0.119934, 0.517447, 0.280189, 0.295209, -0.128109, -0.301298, 0.539822, -0.096016, -0.253774, 0.194507, 0.136900, -0.132318, -0.216668, -0.085674, -0.110360, 0.537772, -0.245333, 0.032601, -0.181540, -0.144376, -0.462822, -0.519044, 0.003142, 0.496157, 0.314684, 0.160240, 0.308515, 0.071996, -0.591869, -0.127334, 0.199358, 0.488650, -0.569913, 0.324262, 0.028376, 0.328832, -0.626706, 0.032348, 0.607194, 0.282018, 0.347948, -0.199523];
    bias_2 : ARRAY[0..7] OF REAL := [-0.285531, -0.475641, -0.175878, 0.019417, -0.573957, -0.778474, -0.512658, -0.658435];

    weights_3 : ARRAY[0..63] OF REAL := [-0.052644, 0.066374, 0.269461, 0.070147, 0.191043, 0.353183, 0.526321, 0.097288, -0.306424, 0.359882, -0.366379, 0.457526, -0.314496, 0.424671, -0.567451, -0.261200, -0.063903, -0.100702, 0.038101, -0.359638, 0.039945, 0.308035, -0.256331, 0.113381, -0.309424, -0.469852, 0.232786, -0.404988, 0.022612, -0.523618, 0.226663, -0.215717, -0.549358, 0.152122, 0.545194, -0.046838, 0.473015, -0.289375, -0.512408, 0.140085, -0.201061, -0.036578, 0.554413, 0.464440, -0.352369, 0.134818, 0.143860, 0.490836, -0.079075, 0.360692, -0.466489, 0.247123, 0.442202, 0.516491, -0.368177, 0.488731, -0.394521, 0.384025, -0.255241, 0.248161, 0.197454, -0.285728, -0.204243, -0.311302];
    bias_3 : ARRAY[0..7] OF REAL := [0.000000, -0.303888, -0.504215, -0.632133, -0.204132, -0.012793, -0.219929, -0.178265];

    weights_4 : ARRAY[0..63] OF REAL := [-0.372153, -0.488993, 0.322207, 0.240118, -0.429187, 0.471674, 0.391840, -0.579532, 0.321415, -0.538890, 0.132752, 0.073944, -0.123694, 0.694431, -0.269960, 0.087844, -0.126521, 0.341294, -0.070244, 0.173532, -0.005624, 0.344665, 0.169546, 0.484228, 0.152758, -0.183956, 0.602844, 0.067450, -0.006641, -0.330285, -0.233587, 0.287266, 0.101863, -0.457850, 0.106928, 0.296401, 0.214952, -0.402940, 0.061645, -0.221250, -0.230949, -0.557260, 0.097835, -0.320289, 0.378542, 0.069630, -0.445657, 0.513073, -0.352412, 0.506039, 0.165290, -0.235276, 0.303806, 0.668099, -0.402635, -0.280692, 0.631382, -0.044422, -0.287416, 0.221539, -0.052976, -0.056548, -0.250608, 0.227349];
    bias_4 : ARRAY[0..7] OF REAL := [-0.103465, -0.012799, -0.162917, -0.052841, -0.074329, 0.012691, -0.165048, -0.203017];

    weights_5 : ARRAY[0..63] OF REAL := [0.350090, 0.478327, 0.322544, 0.212199, -0.357885, -0.139371, -0.232106, -0.173757, 0.075121, 0.352410, 0.160664, 0.249571, 0.518267, 0.514736, -0.015430, -0.440535, -0.074149, -0.097590, 0.009644, 0.384010, 0.116925, 0.351556, 0.338084, -0.010518, 0.102964, 0.021784, -0.459467, 0.649173, 0.549041, -0.031172, -0.248861, -0.318134, 0.173310, 0.602255, 0.388658, -0.352535, 0.564807, 0.628043, -0.065580, -0.069271, 0.163177, 0.131918, -0.453420, -0.260330, 0.231469, -0.165007, 0.251804, 0.372251, 0.156891, -0.021854, -0.087787, -0.337316, 0.383704, -0.334202, 0.438766, 0.441235, 0.067210, 0.318544, 0.393558, 0.628349, -0.221055, -0.201679, 0.002116, 0.157983];
    bias_5 : ARRAY[0..7] OF REAL := [0.002347, -0.016679, -0.006121, 0.016294, 0.001573, -0.020066, -0.004888, -0.082204];

    weights_6 : ARRAY[0..63] OF REAL := [0.467065, -0.156833, 0.041059, -0.150482, -0.108769, 0.139341, 0.091010, 0.596164, 0.064976, -0.242640, 0.267655, 0.314285, 0.313145, 0.056125, 0.476261, -0.331380, 0.032076, 0.066871, -0.371934, 0.218925, 0.185759, 0.085391, 0.658773, -0.027300, -0.428536, 0.321574, -0.090949, -0.507993, -0.021525, 0.152182, -0.074321, 0.094513, 0.338598, -0.082085, 0.551722, -0.398247, 0.410017, -0.325104, 0.430805, 0.155829, -0.451561, -0.569867, 0.176546, -0.210668, 0.116334, 0.462507, 0.312571, 0.579973, -0.387810, 0.187643, 0.403673, -0.064323, -0.062442, 0.185692, 0.779162, 0.177727, 0.483648, 0.054514, 0.608699, 0.278995, -0.157162, -0.047183, 0.051780, -0.111305];
    bias_6 : ARRAY[0..7] OF REAL := [-0.005969, -0.007131, 0.004142, -0.013770, 0.002106, -0.006670, -0.003984, 0.000646];

    weights_7 : ARRAY[0..63] OF REAL := [0.203861, -0.030972, 0.333219, -0.456117, -0.394599, 0.303750, -0.175437, 0.256127, -0.065839, -0.080769, -0.340820, -0.465902, -0.267402, 0.275411, 0.412801, 0.466712, 0.552644, 0.205115, -0.386721, -0.547780, -0.305723, 0.047039, 0.331036, -0.266380, 0.455183, 0.230124, -0.192046, 0.235310, -0.144356, 0.084877, 0.051110, 0.190368, 0.128007, 0.595271, 0.241468, -0.303561, 0.586221, 0.226603, -0.216575, -0.350460, 0.545203, 0.524606, -0.398826, -0.663746, 0.009908, 0.298770, 0.535066, 0.078847, -0.388545, 0.451353, 0.464207, -0.215806, -0.341532, -0.359186, 0.243410, 0.498955, -0.202738, 0.239711, 0.416047, -0.548960, 0.615408, -0.138862, -0.029144, 0.434748];
    bias_7 : ARRAY[0..7] OF REAL := [0.002285, -0.000741, 0.000816, -0.122510, -0.003992, -0.003720, 0.001075, -0.003060];

    weights_8 : ARRAY[0..63] OF REAL := [-0.046600, -0.086008, 0.643339, 0.744063, -0.001908, -0.173786, -0.109752, -0.073092, -0.372336, -0.098538, 0.218392, 0.178496, 0.274282, 0.356771, -0.168973, -0.400447, 0.479468, 0.084380, 0.020090, -0.071978, 0.313519, -0.345538, 0.380101, -0.587423, -0.316940, 0.190187, -0.300594, -0.392995, 0.351047, -0.009114, 0.138731, 0.291449, 0.003388, 0.437885, -0.072545, -0.303327, 0.389802, 0.309439, -0.364275, -0.705197, 0.532831, -0.267534, 0.014498, 0.447030, 0.570693, 0.086147, 0.215370, -0.747437, 0.493814, 0.572020, -0.092239, -0.288292, 0.220241, -0.156123, 0.087341, -0.620701, 0.155317, -0.246157, 0.478788, 0.541892, -0.406391, -0.010187, 0.135038, -0.623599];
    bias_8 : ARRAY[0..7] OF REAL := [0.004908, -0.000114, 0.001135, 0.000904, 0.007861, 0.001130, 0.000515, 0.200354];

    weights_9 : ARRAY[0..63] OF REAL := [-0.061378, 0.256985, 0.148553, 0.333983, -0.279352, -0.139097, 0.339744, 0.267641, 0.327265, 0.245748, 0.504522, 0.238158, -0.367604, 0.381190, 0.557895, 0.168014, 0.291891, -0.696233, -0.349165, 0.250336, -0.367697, 0.359604, 0.232180, 0.200219, -0.110292, 0.227855, 0.548814, -0.074591, -0.569009, 0.072527, 0.339889, 0.228495, -0.278042, 0.167290, 0.454097, 0.325023, -0.003931, -0.140063, 0.056050, 0.525010, 0.279004, 0.420137, -0.035831, 0.373170, -0.026086, 0.436152, 0.153678, -0.339207, 0.226397, 0.484994, 0.096307, -0.305389, 0.021887, 0.484001, -0.076286, 0.174181, -0.356453, -0.125135, -0.418990, -0.660315, -0.203342, -0.704165, -0.612714, -0.622012];
    bias_9 : ARRAY[0..7] OF REAL := [0.003649, 0.004185, 0.085452, 0.145365, -0.158122, 0.154411, 0.132190, 0.084785];

    weights_10 : ARRAY[0..63] OF REAL := [0.396305, 0.297458, -0.167428, 0.118225, -0.008989, 0.643233, 0.685896, 0.440837, 0.519786, 0.158835, 0.143500, 0.018256, 0.133496, 0.374514, 0.318299, -0.023356, 0.376109, 0.151008, -0.336215, -0.487064, -0.234471, -0.027382, 0.388061, -0.124971, 0.212901, 0.434121, -0.454293, -0.313134, 0.073076, -0.108580, 0.361257, 0.477278, -0.386355, 0.028752, 0.138439, 0.212546, -0.481623, -0.021771, -0.445869, 0.280399, 0.341589, 0.614036, -0.118696, -0.715768, -0.161513, -0.191181, 0.538065, 0.094913, 0.461094, 0.224977, -0.678048, -0.524899, -0.625924, 0.026496, 0.037134, 0.308609, 0.293745, 0.536145, -0.174704, -0.036950, -0.523137, 0.229579, -0.155009, 0.260998];
    bias_10 : ARRAY[0..7] OF REAL := [-0.001267, -0.000033, -0.342426, -0.259913, -0.462436, -0.261314, 0.000276, 0.002726];

    weights_11 : ARRAY[0..23] OF REAL := [-0.494317, 0.207545, 0.336739, -0.791353, -0.260368, -0.122563, -0.431979, 0.247782, -0.376800, 0.187500, 0.410269, -0.339999, -0.085222, 0.410256, -0.217633, -0.090285, -0.539762, 0.197141, -0.625611, 0.275213, 0.472093, -0.920704, -0.471168, -0.270643];
    bias_11 : ARRAY[0..2] OF REAL := [1.217250, -0.268151, -0.804870];

END_VAR

VAR
    (* Buffer allocation variables *)
    buffer_0 : ARRAY[0..7] OF REAL;
    buffer_1 : ARRAY[0..7] OF REAL;

    (* Temporary computation variables *)
    i : DINT;
    j : DINT;
    sum : REAL;
    max_val : REAL;
    exp_sum : REAL;

END_VAR

(* Layer 0: Fused Linear + RELU *)
FOR j := 0 TO 7 DO
    sum := 0.0;
    FOR i := 0 TO 4 DO
        sum := sum + input_data[i] * weights_0[i * 8 + j];
    END_FOR;
    buffer_1[j] := MAX(sum + bias_0[j], 0.0);
END_FOR;

(* Layer 1: Fused Linear + RELU *)
FOR j := 0 TO 7 DO
    sum := 0.0;
    FOR i := 0 TO 7 DO
        sum := sum + buffer_1[i] * weights_1[i * 8 + j];
    END_FOR;
    buffer_0[j] := MAX(sum + bias_1[j], 0.0);
END_FOR;

(* Layer 2: Fused Linear + RELU *)
FOR j := 0 TO 7 DO
    sum := 0.0;
    FOR i := 0 TO 7 DO
        sum := sum + buffer_0[i] * weights_2[i * 8 + j];
    END_FOR;
    buffer_1[j] := MAX(sum + bias_2[j], 0.0);
END_FOR;

(* Layer 3: Fused Linear + RELU *)
FOR j := 0 TO 7 DO
    sum := 0.0;
    FOR i := 0 TO 7 DO
        sum := sum + buffer_1[i] * weights_3[i * 8 + j];
    END_FOR;
    buffer_0[j] := MAX(sum + bias_3[j], 0.0);
END_FOR;

(* Layer 4: Fused Linear + RELU *)
FOR j := 0 TO 7 DO
    sum := 0.0;
    FOR i := 0 TO 7 DO
        sum := sum + buffer_0[i] * weights_4[i * 8 + j];
    END_FOR;
    buffer_1[j] := MAX(sum + bias_4[j], 0.0);
END_FOR;

(* Layer 5: Fused Linear + RELU *)
FOR j := 0 TO 7 DO
    sum := 0.0;
    FOR i := 0 TO 7 DO
        sum := sum + buffer_1[i] * weights_5[i * 8 + j];
    END_FOR;
    buffer_0[j] := MAX(sum + bias_5[j], 0.0);
END_FOR;

(* Layer 6: Fused Linear + RELU *)
FOR j := 0 TO 7 DO
    sum := 0.0;
    FOR i := 0 TO 7 DO
        sum := sum + buffer_0[i] * weights_6[i * 8 + j];
    END_FOR;
    buffer_1[j] := MAX(sum + bias_6[j], 0.0);
END_FOR;

(* Layer 7: Fused Linear + RELU *)
FOR j := 0 TO 7 DO
    sum := 0.0;
    FOR i := 0 TO 7 DO
        sum := sum + buffer_1[i] * weights_7[i * 8 + j];
    END_FOR;
    buffer_0[j] := MAX(sum + bias_7[j], 0.0);
END_FOR;

(* Layer 8: Fused Linear + RELU *)
FOR j := 0 TO 7 DO
    sum := 0.0;
    FOR i := 0 TO 7 DO
        sum := sum + buffer_0[i] * weights_8[i * 8 + j];
    END_FOR;
    buffer_1[j] := MAX(sum + bias_8[j], 0.0);
END_FOR;

(* Layer 9: Fused Linear + RELU *)
FOR j := 0 TO 7 DO
    sum := 0.0;
    FOR i := 0 TO 7 DO
        sum := sum + buffer_1[i] * weights_9[i * 8 + j];
    END_FOR;
    buffer_0[j] := MAX(sum + bias_9[j], 0.0);
END_FOR;

(* Layer 10: Fused Linear + RELU *)
FOR j := 0 TO 7 DO
    sum := 0.0;
    FOR i := 0 TO 7 DO
        sum := sum + buffer_0[i] * weights_10[i * 8 + j];
    END_FOR;
    buffer_1[j] := MAX(sum + bias_10[j], 0.0);
END_FOR;

(* Layer 11: Fused Linear + SOFTMAX *)
FOR j := 0 TO 2 DO
    sum := 0.0;
    FOR i := 0 TO 7 DO
        sum := sum + buffer_1[i] * weights_11[i * 3 + j];
    END_FOR;
    output_data[j] := sum + bias_11[j];
END_FOR;

max_val := output_data[0];
FOR i := 1 TO 2 DO
    IF output_data[i] > max_val THEN
        max_val := output_data[i];
    END_IF;
END_FOR;

exp_sum := 0.0;
FOR i := 0 TO 2 DO
    output_data[i] := EXP(output_data[i] - max_val);
    exp_sum := exp_sum + output_data[i];
END_FOR;

FOR i := 0 TO 2 DO
    output_data[i] := output_data[i] / exp_sum;
END_FOR;

END_FUNCTION_BLOCK
